*)
METHOD instantSort : CNM_CollectionInterfaces.CNM_ReturnTypes.SingleExecutionResult
VAR_INPUT
	(*The size of the list to be sorted*)
	size	: UDINT;
	(*Optional: the comparator that should be used for the sort. Must not be changed while sort is in process*)
	comparator	: CNM_CollectionInterfaces.CNM_AbstractObject.IComparator := 0;
END_VAR
VAR_IN_OUT
	(*The first element in the list, must be set on every call to current head of list.*)
	head	: CNM_CollectionInterfaces.IDoublyLinkedElement;
	(*The last element of the list after sorting, may be useful for doublelinked structures*)
	last	: CNM_CollectionInterfaces.IDoublyLinkedElement;
	(*the current version of the list, must change when the data in the list changes *)
	currentListVersion	: __XWORD;
END_VAR
VAR
	mergesThisRun 		:__XWORD;
	mergeSize			:__XWORD;
	mergeSizeLeft		:__XWORD;
	mergeSizeRight		:__XWORD;
	index				:__XWORD;
	leftElementToMerge	:CNM_CollectionInterfaces.IDoublyLinkedElement;
	rightElementToMerge	:CNM_CollectionInterfaces.IDoublyLinkedElement;
	sortComplete :BOOL := FALSE;
	comparesThisCycle	:__XWORD := 0;
END_VAR
VAR CONSTANT
	OBJECT_NOT_REFERENCED 	:__XWORD := 0;
END_VAR
THIS^.sorterHead := head;
THIS^.sorterLast := OBJECT_NOT_REFERENCED;
THIS^.setComparator(comparator);
mergeSize := 1;
WHILE NOT sortComplete DO
	IF THIS^.isObjectNull(leftElementToMerge) THEN 
		mergesThisRun := 0;	
		leftElementToMerge := THIS^.sorterHead;	
		THIS^.sorterHead := OBJECT_NOT_REFERENCED;
		THIS^.sorterLast := OBJECT_NOT_REFERENCED;		
	END_IF;
		
	//one run trought the list from left to right
	WHILE THIS^.isObjectValid(leftElementToMerge) DO
		mergesThisRun := mergesThisRun + 1;
		rightElementToMerge := leftElementToMerge;
		//place rightElement mergeSize steps right of leftElement
		mergeSizeLeft := 0;	
		FOR index := 0 TO mergeSize-1 DO
			mergeSizeLeft := mergeSizeLeft + 1;
			rightElementToMerge := rightElementToMerge.next;
			IF THIS^.isObjectNull(rightElementToMerge) THEN
				EXIT;
			END_IF
		END_FOR
		mergeSizeRight := mergeSize;
		
		THIS^.merge(	
			leftElement := leftElementToMerge,
			rightElement := rightElementToMerge,
			mergeSizeLeft := mergeSizeLeft,
			mergeSizeRight := mergeSizeRight,
			mergeHead := THIS^.sorterHead,
			mergeLast := THIS^.sorterLast,
			comparesThisCycle := comparesThisCycle
		);
		
		//set leftElementToMerge to first unmerged Element, as rightElementToMerge points to the Element behind the right Mergesection
		leftElementToMerge := rightElementToMerge;
	END_WHILE
	
	IF (mergesThisRun <= 1) AND THIS^.isObjectNull(leftElementToMerge) THEN
		sortComplete := TRUE;
	ELSIF THIS^.isObjectNull(leftElementToMerge) THEN
		mergeSize := mergeSize * 2;
	END_IF;
	
	head := THIS^.sorterHead;
	last := THIS^.sorterLast;

END_WHILE

currentListVersion := currentListVersion + 1;
instantSort := CNM_ReturnTypes.SingleExecutionResult.SUCCESS;
END_METHOD

(*

## Short summary

Does an inplace ordered Merge of two list sections, that are defined by their first object and the length of the section.
Merge is achived by updating the links of the elements.

.. <legal notes>

legal notes
=================
| SPDX-FileCopyrightText: © 2024 ekvip automation GmbH <info@ekvip.de>
| SPDX-License-Identifier: Apache-2.0
| For details check: Apache-2.0_

.. _Apache-2.0: https://www.apache.org/licenses/LICENSE-2.0

.. </legal notes>


**Return:** CNM_ReturnTypes.ExecutionState: the state of the merge, 
	SUCCESS if list is merged from left to right bound, 
	BUSY if list not completly merged, needs to be called again.

*)

METHOD PROTECTED merge
VAR_INPUT
	//how many elements are in the left section
	mergeSizeLeft 	:__XWORD;
	//how many elements are in the right section
	mergeSizeRight	:__XWORD;
END_VAR
VAR_IN_OUT
	//The updated head of the list that is beeing merged
	mergeHead			:CNM_CollectionInterfaces.IDoublyLinkedElement;
	//The updated last of the list that is beeing merged
	mergeLast			:CNM_CollectionInterfaces.IDoublyLinkedElement;
	//the first element of the left section
	leftElement			:CNM_CollectionInterfaces.IDoublyLinkedElement;
	// the first element of the right section
	rightElement		:CNM_CollectionInterfaces.IDoublyLinkedElement;
	//The amount of already performed compares this cycle
	comparesThisCycle :__XWORD;
END_VAR
VAR
	remainElementsLeft	:__XWORD := mergeSizeLeft;
	remainElementsRight	:__XWORD := mergeSizeRight;
	elementToMerge		:CNM_CollectionInterfaces.IDoublyLinkedElement;
	lastLeftElement	:CNM_CollectionInterfaces.IDoublyLinkedElement;
END_VAR
VAR CONSTANT
	OBJECT_NOT_REFERENCED :__XWORD := 0;
END_VAR
IF THIS^.isObjectValid(rightElement) THEN
	lastLeftElement := rightElement.previous;	
END_IF

//when remainElementsRight is greater 0, also check if currentRightElement is valid, may not be valid for the merge at end of the list
WHILE(remainElementsLeft > 0 AND_THEN remainElementsRight > 0 AND_THEN THIS^.isObjectValid(rightElement) ) DO
	//by comparing that way, when elements are equal, they are taken from left, making the sort Stable 
	IF THIS^.compareElements(rightElement.object,leftElement.object) = CNM_ReturnTypes.ComparationResult.SMALLER THEN
		elementToMerge := rightElement;
		rightElement := rightElement.next;
		remainElementsRight := remainElementsRight - 1;
	ELSE
		elementToMerge := leftElement;
		leftElement := leftElement.next;
		remainElementsLeft := remainElementsLeft - 1;
	END_IF;
	
	IF THIS^.isObjectNull(mergeHead) THEN
		mergeHead := elementToMerge;
	ELSE
		mergeLast.next := elementToMerge;
	END_IF;
	
	elementToMerge.previous := mergeLast;	
	mergeLast := elementToMerge;
	comparesThisCycle := comparesThisCycle+1;
END_WHILE

elementToMerge := SEL(
	remainElementsLeft > 0,
	rightElement,
	leftElement
);
moveRemainingElements(
	remainingElements := SEL(
		remainElementsLeft > 0,
		remainElementsRight,
		remainElementsLeft
	),
	elementToMerge := elementToMerge,
	mergeHead := mergeHead,
	mergeLast := mergeLast,
	lastRemainder := SEL(remainElementsLeft>0,OBJECT_NOT_REFERENCED,lastLeftElement),
	operationsCount := comparesThisCycle
);	

IF remainElementsRight > 0 AND_THEN THIS^.isObjectValid(rightElement) THEN
	rightElement := mergeLast.next;
ELSE
	mergeLast.next := rightElement;
END_IF

IF THIS^.isObjectValid(rightElement) THEN
	rightElement.previous := mergeLast;	
END_IF
END_METHOD

METHOD moveRemainingElements : BOOL
VAR_INPUT
	remainingElements :__XWORD;
	lastRemainder	:CNM_CollectionInterfaces.IDoublyLinkedElement;
END_VAR
VAR_IN_OUT
	elementToMerge	:CNM_CollectionInterfaces.IDoublyLinkedElement;
	mergeHead		:CNM_CollectionInterfaces.IDoublyLinkedElement;
	mergeLast		:CNM_CollectionInterfaces.IDoublyLinkedElement;
	
	operationsCount	:__XWORD;
END_VAR
//one side is empty, other needs to be "copied"
IF THIS^.isObjectNull(mergeHead) THEN
	mergeHead := elementToMerge;
ELSE
	mergeLast.next := elementToMerge;
END_IF;

elementToMerge.previous := mergeLast;	

IF THIS^.isObjectValid(lastRemainder) THEN
	// first and last of the remaining elements are know, so just move the whole section
	mergeLast := lastRemainder;
	operationsCount := operationsCount + 1;
ELSE
	//step over the leftover elements to figure out the last element of that section
	WHILE remainingElements > 0 AND_THEN THIS^.isObjectValid(elementToMerge) DO
		mergeLast := elementToMerge;	
		elementToMerge := elementToMerge.next;
		remainingElements := remainingElements - 1;
		operationsCount := operationsCount +1;
	END_WHILE
END_IF
END_METHOD

(*

## Short summary

This method sorts the data structure. 
It uses the passed Comperator to sort the structure.
This can take many cycles and should be called until the CNM_ReturnTypes.ExecutionState is no longer ``BUSY``.

.. <legal notes>

legal notes
=================
| SPDX-FileCopyrightText: © 2025 ekvip automation GmbH <info@ekvip.de>
| SPDX-License-Identifier: Apache-2.0
| For details check: Apache-2.0_

.. _Apache-2.0: https://www.apache.org/licenses/LICENSE-2.0

.. </legal notes>


**Return:** ``ABORTED``: While sort was pending,execute had a falling edge,
	``BUSY``: Sort is in progress
	``ERROR``: Sort was not able to finish (p.e. List changed) call sort(false) to reset
	``IDLE``: Currently no sort in progress
	``SUCCESS``: Sorting was finished 

*)
METHOD sort : CNM_ReturnTypes.SingleExecutionState
VAR_INPUT
	(*control bit to start or abort the sorting, needs to be active until the ExecutionState is SUCCESS*)
	execute	: BOOL;
	(*The size of the list to be sorted*)
	size :UDINT;
	(*the comparator that should be used for the sort. Must not be changed while sort is in process*)
	comparator	: CNM_AbstractObject.IComparator	:= 0;
END_VAR
VAR_IN_OUT
	(*The first element in the list, must be set on every call to current head of list.*)
	head :CNM_CollectionInterfaces.IDoublyLinkedElement;
	(*The last element of the list after sorting, may be useful for doublelinked structures*)
	last :CNM_CollectionInterfaces.IDoublyLinkedElement;
	(*the current version of the list, must change when the data in the list changes *)
	currentListVersion :__XWORD;
END_VAR
VAR_INST
	cycleManager 		:CNM_CycleManager.SimpleCycleManager;
	leftElementToMerge	:CNM_CollectionInterfaces.IDoublyLinkedElement;
	rightElementToMerge	:CNM_CollectionInterfaces.IDoublyLinkedElement;
	(*How many merges were made during traversing list from left to right*)
	mergesThisRun 		:__XWORD;
	mergeSize			:__XWORD;
	mergeSizeLeft		:__XWORD;
	mergeSizeRight		:__XWORD;
	index				:__XWORD;
	(* list version index, used to detect list changes during sorting *)
	lastListChangeIndex :__XWORD;
END_VAR
VAR
	comparesThisCycle	:__XWORD	:= 0;
END_VAR
VAR CONSTANT
	INIT	:DINT := CNM_ReturnTypes.DefaultSteps.STEP.INIT; 
	SUCCESS :DINT := CNM_ReturnTypes.DefaultSteps.STEP.SUCCESS;
	ERROR   :DINT := CNM_ReturnTypes.DefaultSteps.STEP.ERROR;
	RUN_SORT :DINT := INIT + 1;
	OBJECT_NOT_REFERENCED 	:__XWORD := 0;
END_VAR
cycleManager(execute := execute);
IF cycleManager.step.current > INIT THEN
	cycleManager.assert.bitNumber.x.valueIsEqualTo(
		currentValue := currentListVersion,
		expectedValue := lastListChangeIndex,
		message := 'List has changed during sort!'
	);
END_IF

CASE cycleManager.step.current OF
INIT:
	cycleManager.configuration.sequence.requireSuccessStep := FALSE;
	lastListChangeIndex := currentListVersion;
	THIS^.sorterHead := head;
	THIS^.sorterLast := OBJECT_NOT_REFERENCED;
	THIS^.setComparator(comparator);
	mergeSize := 1;
	cycleManager.proceedWith(
		step := SEL( (size > 1), SUCCESS, RUN_SORT)
	);
RUN_SORT:
	IF (currentListVersion <> lastListChangeIndex) THEN
		cycleManager.proceedWith(ERROR);
		sort := CNM_ReturnTypes.SingleExecutionState.ERROR;
		RETURN;
	ELSE
		IF THIS^.isObjectNull(leftElementToMerge) THEN 
			mergesThisRun := 0;	
			leftElementToMerge := THIS^.sorterHead;	
			THIS^.sorterHead := OBJECT_NOT_REFERENCED;
			THIS^.sorterLast := OBJECT_NOT_REFERENCED;		
		END_IF;
		
		//one run trought the list from left to right
		WHILE THIS^.isObjectValid(leftElementToMerge) DO
			//only do merge if it won't exceed comparelimit, but allow at least one merge per Cycle
			IF (comparesThisCycle > 0) AND_THEN (comparesThisCycle + mergeSizeLeft + mergeSizeRight > THIS^.upperCompareBound) THEN
				EXIT;
			END_IF
			mergesThisRun := mergesThisRun + 1;
			rightElementToMerge := leftElementToMerge;
			//place rightElement mergeSize steps right of leftElement
			mergeSizeLeft := 0;	
			FOR index := 0 TO mergeSize-1 DO
				mergeSizeLeft := mergeSizeLeft + 1;
				rightElementToMerge := rightElementToMerge.next;
				IF THIS^.isObjectNull(rightElementToMerge) THEN
					EXIT;
				END_IF
			END_FOR
			mergeSizeRight := mergeSize;
			
			THIS^.merge(	
				leftElement := leftElementToMerge,
				rightElement := rightElementToMerge,
				mergeSizeLeft := mergeSizeLeft,
				mergeSizeRight := mergeSizeRight,
				mergeHead := THIS^.sorterHead,
				mergeLast := THIS^.sorterLast,
				comparesThisCycle := comparesThisCycle
			);
			
			//set leftElementToMerge to first unmerged Element, as rightElementToMerge points to the Element behind the right Mergesection
			leftElementToMerge := rightElementToMerge;
		END_WHILE
	
		IF (mergesThisRun <= 1) AND THIS^.isObjectNull(leftElementToMerge) THEN
			cycleManager.proceedWith(SUCCESS);
		ELSIF THIS^.isObjectNull(leftElementToMerge) THEN
			mergeSize := mergeSize * 2;
		END_IF;
	
		head := THIS^.sorterHead;
		last := THIS^.sorterLast;
		
		lastListChangeIndex := currentListVersion := currentListVersion + 1;
	END_IF
END_CASE

sort := cycleManager.state;
END_METHOD

END_FUNCTION_BLOCK

// ---- Lists/Sorter/classes/AbstractLinkedListSorter.TcPOU
(*

## Short summary

Abstract base class for LinkedListSorters.
Handles the head and last properties as well as the clone.
.. <legal notes>

legal notes
=================
| SPDX-FileCopyrightText: © 2025 ekvip automation GmbH <info@ekvip.de>
| SPDX-License-Identifier: Apache-2.0
| For details check: Apache-2.0_

.. _Apache-2.0: https://www.apache.org/licenses/LICENSE-2.0

.. </legal notes>



*)

FUNCTION_BLOCK INTERNAL ABSTRACT AbstractLinkedListSorter EXTENDS AbstractListSorter IMPLEMENTS CNM_CollectionInterfaces.ILinkedListSorter
VAR
	sorterHead :CNM_CollectionInterfaces.IDoublyLinkedElement;
	sorterLast :CNM_CollectionInterfaces.IDoublyLinkedElement;
END_VAR

(*

## Short summary

This method sorts the data structure instantly in descending order within one call. 
Uses the passed Comparator or the compareTo of the contained Objects if no comparator is passed.

.. <legal notes>

legal notes
=================
| SPDX-FileCopyrightText: © 2022 ekvip automation GmbH <info@ekvip.de>
| SPDX-License-Identifier: Apache-2.0
| For details check: Apache-2.0_

.. _Apache-2.0: https://www.apache.org/licenses/LICENSE-2.0

.. </legal notes>


**Return:**``ERROR``: Sort was not able to finish 
	``SUCCESS``: Sorting was finished succesfully

*)
METHOD instantInverseSort : CNM_CollectionInterfaces.CNM_ReturnTypes.SingleExecutionResult
VAR_INPUT
	(*The size of the list to be sorted*)
	size	: UDINT;
	(*Optional: the comparator that should be used for the sort. Must not be changed while sort is in process*)
	comparator	: CNM_CollectionInterfaces.CNM_AbstractObject.IComparator := 0;
END_VAR
VAR_IN_OUT
	(*The first element in the list, must be set on every call to current head of list.*)
	head	: CNM_CollectionInterfaces.IDoublyLinkedElement;
	(*The last element of the list after sorting, may be useful for doublelinked structures*)
	last	: CNM_CollectionInterfaces.IDoublyLinkedElement;
	(*the current version of the list, must change when the data in the list changes *)
	currentListVersion	: __XWORD;
END_VAR
THIS^.reverseComparator.attachComparator(comparator);
THIS^.instantSort(
	size := size,
	comparator := THIS^.reverseComparator,
	head := head,
	last := last,
	currentListVersion := currentListVersion
);
END_METHOD

(*

## Short summary

This method sorts the data structure instantly within one call. 
Uses the passed Comparator or the compareTo of the contained Objects if no comparator is passed.

.. <legal notes>

legal notes
=================
| SPDX-FileCopyrightText: © 2022 ekvip automation GmbH <info@ekvip.de>
| SPDX-License-Identifier: Apache-2.0
| For details check: Apache-2.0_

.. _Apache-2.0: https://www.apache.org/licenses/LICENSE-2.0

.. </legal notes>


**Return:**``ERROR``: Sort was not able to finish 
	``SUCCESS``: Sorting was finished succesfully

*)
METHOD ABSTRACT instantSort : CNM_CollectionInterfaces.CNM_ReturnTypes.SingleExecutionResult
VAR_INPUT
	(*The size of the list to be sorted*)
	size	: UDINT;
	(*Optional: the comparator that should be used for the sort. Must not be changed while sort is in process*)
	comparator	: CNM_CollectionInterfaces.CNM_AbstractObject.IComparator := 0;
END_VAR
VAR_IN_OUT
	(*The first element in the list, must be set on every call to current head of list.*)
	head	: CNM_CollectionInterfaces.IDoublyLinkedElement;
	(*The last element of the list after sorting, may be useful for doublelinked structures*)
	last	: CNM_CollectionInterfaces.IDoublyLinkedElement;
	(*the current version of the list, must change when the data in the list changes *)
	currentListVersion	: __XWORD;
END_VAR
END_METHOD

(*

## Short summary

This method sorts the Sortable in the inverted order, so from great to low
.. <legal notes>

legal notes
=================
| SPDX-FileCopyrightText: © 2025 ekvip automation GmbH <info@ekvip.de>
| SPDX-License-Identifier: Apache-2.0
| For details check: Apache-2.0_

.. _Apache-2.0: https://www.apache.org/licenses/LICENSE-2.0

.. </legal notes>


**Return:** ``ABORTED``: While inverse was pending,execute had a falling edge,
	``BUSY``: Inverse is in progress
	``ERROR``: Inverse was not able to finish (p.e. List changed) call inverse(false) to reset
	``IDLE``: Currently invert is not in progress
	``SUCCESS``: Inversing was finished 
*)

METHOD inverseSort :CNM_ReturnTypes.SingleExecutionState;
VAR_INPUT
	(*control bit to start or abort the inverting, needs to be active until the ExecutionState is noz longer busy*)
	execute	:BOOL;
	(*The size of the list to be sorted*)
	size :UDINT;
END_VAR
VAR_INPUT
	(*the comparator that should be used for the sort. Must not be changed while sort is in process*)
	comparator :CNM_AbstractObject.IComparator := 0;
END_VAR
VAR_IN_OUT
	(*The first element in the list, must be set on every call to current head of list.*)
	head :CNM_CollectionInterfaces.IDoublyLinkedElement;
	(*The last element of the list after sorting, may be useful for doublelinked structures*)
	last :CNM_CollectionInterfaces.IDoublyLinkedElement;
	(*the current version of the list, must change when the data in the list changes *)
	currentListVersion :__XWORD;
END_VAR
THIS^.reverseComparator.attachComparator(comparator);
THIS^.sort(
	execute := execute,
	size := size,
	comparator := THIS^.reverseComparator,
	head := head,
	last := last,
	currentListVersion := currentListVersion
);
END_METHOD

(*

## Short summary

This method sorts the data structure. 
This can take many cycles and should be called until the CNM_ReturnTypes.ExecutionState is no longer ``BUSY``.
Call with execute := FALSE to initialize before sort.
.. <legal notes>

legal notes
=================
| SPDX-FileCopyrightText: © 2022 ekvip automation GmbH <info@ekvip.de>
| SPDX-License-Identifier: Apache-2.0
| For details check: Apache-2.0_

.. _Apache-2.0: https://www.apache.org/licenses/LICENSE-2.0

.. </legal notes>


**Return:** ``ABORTED``: While sort was pending,execute had a falling edge,
	``BUSY``: Sort is in progress
	``ERROR``: Sort was not able to finish (p.e. List changed) call sort(false) to reset
	``IDLE``: Currently no sort in progress
	``SUCCESS``: Sorting was finished 

*)

METHOD ABSTRACT sort :CNM_ReturnTypes.SingleExecutionState
VAR_INPUT
	(*control bit to start or abort the sorting, needs to be active until the ExecutionState is SUCCESS*)
	execute	:BOOL;
	(*The size of the list to be sorted*)
	size :UDINT;
	(*Optional: the comparator that should be used for the sort. Must not be changed while sort is in process*)
	comparator :CNM_AbstractObject.IComparator := 0;
END_VAR
VAR_IN_OUT
	(*The first element in the list, must be set on every call to current head of list.*)
	head :CNM_CollectionInterfaces.IDoublyLinkedElement;
	(*The last element of the list after sorting, may be useful for doublelinked structures*)
	last :CNM_CollectionInterfaces.IDoublyLinkedElement;
	(*the current version of the list, must change when the data in the list changes *)
	currentListVersion :__XWORD;
END_VAR
END_METHOD

END_FUNCTION_BLOCK

// ---- Utils/log2.TcPOU
(*

## Short summary

This function calculates the logarithmus dualis (ld or log_2). 
It uses [black magic](https://en.wikipedia.org/wiki/De_Bruijn_sequence). Actually it calculates the log2 and truncates it. 

.. <legal notes>

legal notes
=================
| SPDX-FileCopyrightText: © 2025 ekvip automation GmbH <info@ekvip.de>
| SPDX-License-Identifier: Apache-2.0
| For details check: Apache-2.0_

.. _Apache-2.0: https://www.apache.org/licenses/LICENSE-2.0

.. </legal notes>

*)

FUNCTION log2 : USINT
VAR_INPUT
	value :__UXINT(1..MAX_UXINT);
END_VAR
VAR
	architectureIndex :__XWORD;
	registerSize :USINT;
END_VAR
VAR CONSTANT
	MAX_UXINT :__UXINT := TO___UXINT(-1);
	DE_BRUIJN_SEQUENCE	:ARRAY[0..2] OF LWORD := [16#09AF ,16#077CB531, 16#022FDD63CC95386D];
	REGISTER_SIZE_IN_BYTES	:USINT := SIZEOF(__XWORD);
	DE_BRUIJN_LOOKUP :ARRAY[0..2] OF ARRAY[0..63] OF USINT := [
		[
			0, 1, 10, 2, 11, 14, 7, 3, 
        	12, 15, 8, 6, 13, 9, 5, 4
		],
		[
	    	0,  1, 28,  2, 29, 14, 24,  3, 
	    	30, 22, 20, 15, 25, 17,  4,  8, 
	    	31, 27, 13, 23, 21, 19, 16,  7, 
		    26, 12, 18,  6, 11,  5, 10,  9	
		],
		[
			0,  1,  2, 53,  3,  7, 54, 27,
			4, 38, 41,  8, 34, 55, 48, 28,
			62,  5, 39, 46, 44, 42, 22,  9,
			24, 35, 59, 56, 49, 18, 29, 11,
			63, 52,  6, 26, 37, 40, 33, 47,
			61, 45, 43, 21, 23, 58, 17, 10,
			51, 25, 36, 32, 60, 20, 57, 16,
			50, 31, 19, 15, 30, 14, 13, 12		
		]
	];
END_VAR

log2 := TO_USINT(-1);
RETURN(value <= 0);
architectureIndex := SHR(REGISTER_SIZE_IN_BYTES,2);
registerSize := SHL(REGISTER_SIZE_IN_BYTES,3);
value := value OR SHR(value, 1);
value := value OR SHR(value, 2);
value := value OR SHR(value, 4);
value := value OR SHR(value, 8);
value := SEL((REGISTER_SIZE_IN_BYTES > 2), value, (value OR SHR(value, 16)));
value := SEL((REGISTER_SIZE_IN_BYTES > 4), value, (value OR SHR(value, 32)));
IF (value = MAX_UXINT) THEN
	log2 := registerSize - 1;
ELSE
	log2 := DE_BRUIJN_LOOKUP[architectureIndex][
		SHR((value + 1) * DE_BRUIJN_SEQUENCE[architectureIndex],registerSize - (4 + architectureIndex))
	] - 1;
END_IF

END_FUNCTION

// ---- BinaryTree/Set/SetStrategyExecutor.TcPOU
FUNCTION_BLOCK INTERNAL SetStrategyExecutor EXTENDS CNM_AbstractObject.Object IMPLEMENTS CNM_CollectionInterfaces.ISetStrategy
VAR
	set :ISetHelper;
	instantExecutor :InstantSetStrategyExecutor;
END_VAR

(*

## Short summary

This abstract property returns the class name of the concrete object, 
which is useful for logging/debugging purpose.

.. <legal notes>

legal notes
=================
| SPDX-FileCopyrightText: © 2022 ekvip automation GmbH <info@ekvip.de>
| SPDX-License-Identifier: Apache-2.0
| For details check: Apache-2.0_

.. _Apache-2.0: https://www.apache.org/licenses/LICENSE-2.0

.. </legal notes>

*)
PROPERTY className : CNM_AbstractObject.ClassName
GET
className := 'CNM_Collections.SetStrategyExecutor';
END_GET
END_PROPERTY

(*

## Short summary

The constructor ``FB_init`` is needed to create an unique hash code.
The hash code is a pseudo random number create with a [xorshift](https://en.wikipedia.org/wiki/Xorshift) algorithm.
It can be overwritten on derivations, because it will be called implicit, ``SUPER^.FB_init()`` is not required.
For more information check: [Behavoir with derived function blocks](https://infosys.beckhoff.com/content/1033/tc3_plc_intro/5482088715.html?id=6983869892358031022).

.. <legal notes>

legal notes
=================
| SPDX-FileCopyrightText: © 2022 ekvip automation GmbH <info@ekvip.de>
| SPDX-License-Identifier: Apache-2.0
| For details check: Apache-2.0_

.. _Apache-2.0: https://www.apache.org/licenses/LICENSE-2.0

.. </legal notes>



*)
METHOD FB_init : BOOL
VAR_INPUT
	(* if TRUE, the retain variables are initialized (warm start / cold start)*)
	bInitRetains	: BOOL;
	(* if TRUE, the instance afterwards gets moved into the copy code (online change) *)
	bInCopyCode	: BOOL;
	(* the set which this executor will dispatch  *)
	set :ISetHelper;
END_VAR
THIS^.set := set;
THIS^.instantExecutor.assignSet(set);
END_METHOD

(*

## Short summary

Searches an object that is equal to the provided object in terms of the compareTo method (or a comparator provided by the parent).
 
.. <legal notes>

legal notes
=================
| SPDX-FileCopyrightText: © 2023 ekvip automation GmbH <info@ekvip.de>
| SPDX-License-Identifier: Apache-2.0
| For details check: Apache-2.0_

.. _Apache-2.0: https://www.apache.org/licenses/LICENSE-2.0

.. </legal notes>


**Return:** ``TRUE`` when an object that is equal is found, otherwise ``FALSE``

*)
METHOD getEqualObject : BOOL
VAR_INPUT
	(*The object to search for*)
	object	: CNM_CollectionInterfaces.CNM_AbstractObject.IObject;
END_VAR
VAR_OUTPUT
	(*The found object or null if not found*)
	foundObject	: CNM_CollectionInterfaces.CNM_AbstractObject.IObject;
END_VAR
getEqualObject := THIS^.set.getEqualObject(object := object, foundObject => foundObject);
END_METHOD

(*

## Short summary

This property returns a fluent interface for immediate (wihtin one call) operations of sets.

.. <legal notes>

legal notes
=================
| SPDX-FileCopyrightText: © 2025 ekvip automation GmbH <info@ekvip.de>
| SPDX-License-Identifier: Apache-2.0
| For details check: Apache-2.0_

.. _Apache-2.0: https://www.apache.org/licenses/LICENSE-2.0

.. </legal notes>

*)
PROPERTY instant : CNM_CollectionInterfaces.IInstantSetStrategy
GET
instant := THIS^.instantExecutor;
END_GET
END_PROPERTY

(*

## Short summary

overwrites the content of this set with the intersection of this set and the given set
Set intersection: Common elements between two sets.

**Example:**
Set A = {2, 3, 1, 4}
Set B = {3, 5, 6, 4}

Intersection of A and B: {3, 4}

.. <legal notes>

legal notes
=================
| SPDX-FileCopyrightText: © 2022 ekvip automation GmbH <info@ekvip.de>
| SPDX-License-Identifier: Apache-2.0
| For details check: Apache-2.0_

.. _Apache-2.0: https://www.apache.org/licenses/LICENSE-2.0

.. </legal notes>


**Return:** ``SUCCESS``: if intersect is complete
	``ABORTED``: execute has a falling edge during intersect,
	``BUSY``: Intersect is in Progress
	``ERROR``: the passed collection was not valid / contained invalid Elements

*)
METHOD intersect : CNM_CollectionInterfaces.CNM_ReturnTypes.SingleExecutionState
VAR_INPUT
	(*foreign set to intersect with*)
	set	: CNM_CollectionInterfaces.ISet;
	(*If intersect should be processed*)
	execute	: BOOL;
END_VAR
intersect := THIS^.set.intersect(set := set, execute := execute);
END_METHOD

(*

## Short summary

overwrites the content of this set with the union of this set and the given set
Set union: Combination of all elements from two sets.

**Example:**
Set A = {2, 3, 1, 4}
Set B = {3, 5, 6, 4}

Union of A and B: {1, 2, 3, 4, 5, 6}

.. <legal notes>

legal notes
=================
| SPDX-FileCopyrightText: © 2022 ekvip automation GmbH <info@ekvip.de>
| SPDX-License-Identifier: Apache-2.0
| For details check: Apache-2.0_

.. _Apache-2.0: https://www.apache.org/licenses/LICENSE-2.0

.. </legal notes>


**Return:** ``SUCCESS``: if merge completed, 
	``ABORTED``: execute has a falling edge during merge,
	``BUSY``: merge is in Progress
	``ERROR``: the passed collection where not valid / contained invalid Elements

*)
METHOD merge : CNM_CollectionInterfaces.CNM_ReturnTypes.SingleExecutionState
VAR_INPUT
	(*foreign set to merge with*)
	set	: CNM_CollectionInterfaces.ISet;
	(*If merge should be processed*)
	execute	: BOOL;
END_VAR
merge := THIS^.set.merge(set := set, execute := execute);
END_METHOD

(*

## Short summary

overwrites the content of this set with the set difference of this set and the given set
Set difference: Elements present in one set but not in the other.

**Example:**
Set A = {2, 3, 1, 4}
Set B = {3, 5, 6, 4}

Set difference (A - B): {1, 2}
Set difference (B - A): {5, 6}

.. <legal notes>

legal notes
=================
| SPDX-FileCopyrightText: © 2022 ekvip automation GmbH <info@ekvip.de>
| SPDX-License-Identifier: Apache-2.0
| For details check: Apache-2.0_

.. _Apache-2.0: https://www.apache.org/licenses/LICENSE-2.0

.. </legal notes>


**Return:** ``SUCCESS``: if insert could made, error if object was already in the tree,
	``ABORTED``: execute has a falling edge during insert,
	``BUSY``: Insert is in Progress
	``ERROR``: the passed collection where not valid / contained invalid Elements

*)
METHOD subtract : CNM_CollectionInterfaces.CNM_ReturnTypes.SingleExecutionState
VAR_INPUT
	(*foreign set to construct substraction*)
	set	: CNM_CollectionInterfaces.ISet;
	(*If substract should be processed*)
	execute	: BOOL;
END_VAR
subtract := THIS^.set.subtract(set := set, execute := execute);
END_METHOD

END_FUNCTION_BLOCK

// ---- BinaryTree/Set/InstantSetStrategyExecutor.TcPOU
FUNCTION_BLOCK INTERNAL InstantSetStrategyExecutor EXTENDS CNM_AbstractObject.Object IMPLEMENTS CNM_CollectionInterfaces.IInstantSetStrategy
VAR
	set :ISetHelper;
END_VAR

METHOD INTERNAL assignSet
VAR_INPUT
	set :ISetHelper;
END_VAR
THIS^.set := set;
END_METHOD

(*

## Short summary

This abstract property returns the class name of the concrete object, 
which is useful for logging/debugging purpose.

.. <legal notes>

legal notes
=================
| SPDX-FileCopyrightText: © 2022 ekvip automation GmbH <info@ekvip.de>
| SPDX-License-Identifier: Apache-2.0
| For details check: Apache-2.0_

.. _Apache-2.0: https://www.apache.org/licenses/LICENSE-2.0

.. </legal notes>

*)
PROPERTY className : CNM_AbstractObject.ClassName
GET
className := 'CNM_Collections.InstantSetExecutorStrategy';
END_GET
END_PROPERTY

(*

## Short summary

overwrites the content of this set with the intersection of this set and the given set
Set intersection: Common elements between two sets.

**Example:**
Set A = {2, 3, 1, 4}
Set B = {3, 5, 6, 4}

Intersection of A and B: {3, 4}

.. <legal notes>

legal notes
=================
| SPDX-FileCopyrightText: © 2022 ekvip automation GmbH <info@ekvip.de>
| SPDX-License-Identifier: Apache-2.0
| For details check: Apache-2.0_

.. _Apache-2.0: https://www.apache.org/licenses/LICENSE-2.0

.. </legal notes>


**Return:** ``SingleExecutionResult.SUCCESS``: if intersect is complete
	``SingleExecutionResult.ABORTED``: foreign set wasn't valid

*)
METHOD intersect : CNM_CollectionInterfaces.CNM_ReturnTypes.SingleExecutionResult
VAR_INPUT
	(*foreign set to intersect with*)
	set	: CNM_CollectionInterfaces.ISet;
END_VAR
intersect := THIS^.set.instantIntersect(set := set);
END_METHOD

(*

## Short summary

overwrites the content of this set with the union of this set and the given set
Set union: Combination of all elements from two sets.

**Example:**
Set A = {2, 3, 1, 4}
Set B = {3, 5, 6, 4}

Union of A and B: {1, 2, 3, 4, 5, 6}

.. <legal notes>

legal notes
=================
| SPDX-FileCopyrightText: © 2022 ekvip automation GmbH <info@ekvip.de>
| SPDX-License-Identifier: Apache-2.0
| For details check: Apache-2.0_

.. _Apache-2.0: https://www.apache.org/licenses/LICENSE-2.0

.. </legal notes>


**Return:** ``SUCCESS``: if merge completed
	```SingleExecutionResult.ABORTED``: foreign set wasn't valid

*)
METHOD merge : CNM_CollectionInterfaces.CNM_ReturnTypes.SingleExecutionResult
VAR_INPUT
	(*foreign set to merge with*)
	set	: CNM_CollectionInterfaces.ISet;
END_VAR
merge := THIS^.set.instantMerge(set := set);
END_METHOD

(*

## Short summary

overwrites the content of this set with the set difference of this set and the given set
Set difference: Elements present in one set but not in the other.

**Example:**
Set A = {2, 3, 1, 4}
Set B = {3, 5, 6, 4}

Set difference (A - B): {1, 2}
Set difference (B - A): {5, 6}

.. <legal notes>

legal notes
=================
| SPDX-FileCopyrightText: © 2022 ekvip automation GmbH <info@ekvip.de>
| SPDX-License-Identifier: Apache-2.0
| For details check: Apache-2.0_

.. _Apache-2.0: https://www.apache.org/licenses/LICENSE-2.0

.. </legal notes>


**Return:** ``SingleExecutionResult.SUCCESS``: if insert could made, error if object was already in the tree,
	```SingleExecutionResult.ABORTED``: foreign set wasn't valid

*)
METHOD subtract : CNM_CollectionInterfaces.CNM_ReturnTypes.SingleExecutionResult
VAR_INPUT
	(*foreign set to construct substraction*)
	set	: CNM_CollectionInterfaces.ISet;
END_VAR
subtract := THIS^.set.instantSubtract(set := set);
END_METHOD

END_FUNCTION_BLOCK

// ---- BinaryTree/Tree/TreeStrategyExecutor.TcPOU
FUNCTION_BLOCK TreeStrategyExecutor EXTENDS CNM_AbstractObject.Object IMPLEMENTS CNM_CollectionInterfaces.ITreeStrategy
VAR
	tree :ITreeHelper;
	instantExecutor :InstantTreeStrategyExecutor;
END_VAR

(*

## Short summary

This abstract property returns the class name of the concrete object, 
which is useful for logging/debugging purpose.

.. <legal notes>

legal notes
=================
| SPDX-FileCopyrightText: © 2022 ekvip automation GmbH <info@ekvip.de>
| SPDX-License-Identifier: Apache-2.0
| For details check: Apache-2.0_

.. _Apache-2.0: https://www.apache.org/licenses/LICENSE-2.0

.. </legal notes>

*)
PROPERTY className : CNM_AbstractObject.ClassName
GET
className := 'CNM_Collections.TreeStrategyExecutor';
END_GET
END_PROPERTY

(*

## Short summary

The constructor ``FB_init`` is needed to create an unique hash code.
The hash code is a pseudo random number create with a [xorshift](https://en.wikipedia.org/wiki/Xorshift) algorithm.
It can be overwritten on derivations, because it will be called implicit, ``SUPER^.FB_init()`` is not required.
For more information check: [Behavoir with derived function blocks](https://infosys.beckhoff.com/content/1033/tc3_plc_intro/5482088715.html?id=6983869892358031022).

.. <legal notes>

legal notes
=================
| SPDX-FileCopyrightText: © 2022 ekvip automation GmbH <info@ekvip.de>
| SPDX-License-Identifier: Apache-2.0
| For details check: Apache-2.0_

.. _Apache-2.0: https://www.apache.org/licenses/LICENSE-2.0

.. </legal notes>


*)
METHOD FB_init : BOOL
VAR_INPUT
	(* if TRUE, the retain variables are initialized (warm start / cold start)*)
	bInitRetains	: BOOL;
	(* if TRUE, the instance afterwards gets moved into the copy code (online change) *)
	bInCopyCode	: BOOL;
	(*the tree which this executor will dispatch to*)
	tree :ITreeHelper;
END_VAR
THIS^.tree := tree;
THIS^.instantExecutor.assignTree(tree);
END_METHOD

(*

## Short summary

A method to insert a single element into the tree.

.. <legal notes>

legal notes
=================
| SPDX-FileCopyrightText: © 2022 ekvip automation GmbH <info@ekvip.de>
| SPDX-License-Identifier: Apache-2.0
| For details check: Apache-2.0_

.. _Apache-2.0: https://www.apache.org/licenses/LICENSE-2.0

.. </legal notes>


**Return:** ``SUCCESS``: operation successful
	``ABORTED``: operation was aborted (implementation specific)
	``ERROR``: out of memory

*)
METHOD insert : CNM_CollectionInterfaces.CNM_ReturnTypes.SingleExecutionResult
VAR_INPUT
	(*the object that should be inserted*)
	object	: CNM_CollectionInterfaces.CNM_AbstractObject.IObject;
END_VAR
insert := THIS^.tree.insert(object := object);
END_METHOD

(*

## Short summary

This method inserts all elements of a collection into the tree.

If any value of the collection could not be inserted because of duplication, operation isn't aborted, 
insertion is tried for every element of the collection.

.. <legal notes>

legal notes
=================
| SPDX-FileCopyrightText: © 2025 ekvip automation GmbH <info@ekvip.de>
| SPDX-License-Identifier: Apache-2.0
| For details check: Apache-2.0_

.. _Apache-2.0: https://www.apache.org/licenses/LICENSE-2.0

.. </legal notes>


**Return:** ``SUCCESS``: if insert could be made
	``ABORTED``: execute has a falling edge during insert,
	``BUSY``: Insert is in Progress
	``ERROR``: the passed collection where not valid / contained invalid Elements
	``IDLE``: method was never started

*)
METHOD insertCollection : CNM_CollectionInterfaces.CNM_ReturnTypes.SingleExecutionState
VAR_INPUT
	(*The collection that should be inserted*)
	collection	: CNM_CollectionInterfaces.ICollection;
	(*If insert should be processed*)
	execute	: BOOL;
END_VAR
insertCollection := THIS^.tree.insertCollection(collection := collection, execute := execute);
END_METHOD

(*

## Short summary

This property returns a fluent interface for immediate (wihtin one call) operations of tree.

.. <legal notes>

legal notes
=================
| SPDX-FileCopyrightText: © 2025 ekvip automation GmbH <info@ekvip.de>
| SPDX-License-Identifier: Apache-2.0
| For details check: Apache-2.0_

.. _Apache-2.0: https://www.apache.org/licenses/LICENSE-2.0

.. </legal notes>

*)
PROPERTY instant : CNM_CollectionInterfaces.IInstantTreeStrategy
GET
instant := THIS^.instantExecutor;
END_GET
END_PROPERTY

(*

## Short summary

Function to remove an object from the tree

.. <legal notes>

legal notes
=================
| SPDX-FileCopyrightText: © 2022 ekvip automation GmbH <info@ekvip.de>
| SPDX-License-Identifier: Apache-2.0
| For details check: Apache-2.0_

.. _Apache-2.0: https://www.apache.org/licenses/LICENSE-2.0

.. </legal notes>


**Return:** ``SUCCESS``: if remove could be made
	``ABORTED``: if object wasn't in the tree
	``ERROR``: if object wasn't valid

*)
METHOD remove : CNM_CollectionInterfaces.CNM_ReturnTypes.SingleExecutionResult
VAR_INPUT
	(* The object that should be removed *)
	object	: CNM_CollectionInterfaces.CNM_AbstractObject.IObject;
END_VAR
remove := THIS^.tree.remove(object := object);
END_METHOD

END_FUNCTION_BLOCK

// ---- BinaryTree/Tree/InstantTreeStrategyExecutor.TcPOU
FUNCTION_BLOCK InstantTreeStrategyExecutor EXTENDS CNM_AbstractObject.Object IMPLEMENTS CNM_CollectionInterfaces.IInstantTreeStrategy
VAR
	tree :ITreeHelper;
END_VAR

METHOD INTERNAL assignTree
VAR_INPUT
	tree :ITreeHelper;
END_VAR
THIS^.tree := tree;
END_METHOD

(*

## Short summary

This abstract property returns the class name of the concrete object, 
which is useful for logging/debugging purpose.

.. <legal notes>

legal notes
=================
| SPDX-FileCopyrightText: © 2022 ekvip automation GmbH <info@ekvip.de>
| SPDX-License-Identifier: Apache-2.0
| For details check: Apache-2.0_

.. _Apache-2.0: https://www.apache.org/licenses/LICENSE-2.0

.. </legal notes>

*)
PROPERTY className : CNM_AbstractObject.ClassName
GET
className := 'CNM_Collections.InstantTreeStrategyExecutor';
END_GET
END_PROPERTY

(*

## Short summary

This method inserts all elements of a collection into the tree
This takes only one cycle 

.. <legal notes>

legal notes
=================
| SPDX-FileCopyrightText: © 2022 ekvip automation GmbH <info@ekvip.de>
| SPDX-License-Identifier: Apache-2.0
| For details check: Apache-2.0_

.. _Apache-2.0: https://www.apache.org/licenses/LICENSE-2.0

.. </legal notes>


**Return:** ``SingleExecutionResult.SUCCESS``: operation successful
	``SingleExecutionResult.ERROR``: out of memory
	``SingleExecutionResult.ABORTED``: collection to insert wasn't valid

*)
METHOD insertCollection : CNM_CollectionInterfaces.CNM_ReturnTypes.SingleExecutionResult
VAR_INPUT
	(*The collection that should be inserted*)
	collection	: CNM_CollectionInterfaces.ICollection;
END_VAR
insertCollection := THIS^.tree.instantInsertCollection(collection := collection);
END_METHOD

END_FUNCTION_BLOCK

// ---- BinaryTree/classes/BalancedBinarySearchTreeNode.TcPOU
(*

## Short summary

Class for a balanced, binary, search tree node

.. <legal notes>

legal notes
=================
| SPDX-FileCopyrightText: © 2022 ekvip automation GmbH <info@ekvip.de>
| SPDX-License-Identifier: Apache-2.0
| For details check: Apache-2.0_

.. _Apache-2.0: https://www.apache.org/licenses/LICENSE-2.0

.. </legal notes>



*)
{attribute 'enable_dynamic_creation'}
FUNCTION_BLOCK BalancedBinarySearchTreeNode EXTENDS AbstractDisposableContainer IMPLEMENTS CNM_CollectionInterfaces.IBalancedBinarySearchTreeNode
VAR
	nodevalue 			:CNM_AbstractObject.IObject;
	left 				:CNM_CollectionInterfaces.IBinaryTreeNode;
	right				:CNM_CollectionInterfaces.IBinaryTreeNode;
	nodebalance			:CNM_CollectionInterfaces.TreeBalance;
END_VAR

(*

## Short summary

This property represents the balance state for this node, for details see ``Tree_Balance`` from Interfacelib

.. <legal notes>

legal notes
=================
| SPDX-FileCopyrightText: © 2022 ekvip automation GmbH <info@ekvip.de>
| SPDX-License-Identifier: Apache-2.0
| For details check: Apache-2.0_

.. _Apache-2.0: https://www.apache.org/licenses/LICENSE-2.0

.. </legal notes>

*)

PROPERTY balance :CNM_CollectionInterfaces.TreeBalance
GET
balance := THIS^.nodebalance;
END_GET
SET
THIS^.nodebalance := balance;
END_SET
END_PROPERTY


(*

## Short summary

This abstract property returns the class name of the concrete object, 
which is useful to check the class name for ``__DELETE``.

.. <legal notes>

legal notes
=================
| SPDX-FileCopyrightText: © 2022 ekvip automation GmbH <info@ekvip.de>
| SPDX-License-Identifier: Apache-2.0
| For details check: Apache-2.0_

.. _Apache-2.0: https://www.apache.org/licenses/LICENSE-2.0

.. </legal notes>

*)
PROPERTY className :CNM_AbstractObject.ClassName
GET
className := 'CNM_Collections.BalancedBinarySearchTreeNode';
END_GET
END_PROPERTY

(*

## Short summary

This method is called in the destruct method and is intended to zero all references and interfaces that should not be destructed. 
To delete the collection with all its contents, use deepDestruct() instead of destruct().

.. <legal notes>

legal notes
=================
| SPDX-FileCopyrightText: © 2025 ekvip automation GmbH <info@ekvip.de>
| SPDX-License-Identifier: Apache-2.0
| For details check: Apache-2.0_

.. _Apache-2.0: https://www.apache.org/licenses/LICENSE-2.0

.. </legal notes>

*)
METHOD PROTECTED clearContents
VAR CONSTANT
	(* NULL is a constant which is always 0 *)
	NULL						:__XWORD	:= 0;
END_VAR
THIS^.left := NULL;
THIS^.right := NULL;
THIS^.nodevalue := NULL;
END_METHOD


(*

## Short summary

This method is used to create a new instance
of the object which has the same internal state as the object.
If the object is a container class, the content objects
are not cloned, for this there is the method ``ICloneable.deepClone``.

If an object does not support cloning the return value is
``CNM_ReturnTypes.CloneResult.CLONE_IS_NOT_SUPPORTED``.

If there is not enough memory or the cloning fails, because the
attribute enable dynamic creation was forgotten, the return value is 
``CNM_ReturnTypes.CloneResult.FAILED``.

Only if the return value is ``CNM_ReturnTypes.CloneResult.SUCCESS``
the output ``clonedObject`` points to the new object
otherwise ``clonedObject`` is NULL.  

.. <legal notes>

legal notes
=================
| SPDX-FileCopyrightText: © 2022 ekvip automation GmbH <info@ekvip.de>
| SPDX-License-Identifier: Apache-2.0
| For details check: Apache-2.0_

.. _Apache-2.0: https://www.apache.org/licenses/LICENSE-2.0

.. </legal notes>


**Return:** ``CNM_ReturnTypes.CloneResult.SUCCESS``: new object clone was created,
	``CNM_ReturnTypes.CloneResult.FAILED``: object clone failed
	``CNM_ReturnTypes.CloneResult.CLONE_IS_NOT_SUPPORTED``: object does not support cloning

*)
METHOD clone :CNM_AbstractObject.CNM_ReturnTypes.CloneResult
VAR_OUTPUT
	(* new object instance or NULL if somthing went wrong *)
	clonedObject			:CNM_AbstractObject.IObject;
END_VAR
VAR
	newTreeNode 			:POINTER TO BalancedBinarySearchTreeNode;
	newChildObject			:CNM_AbstractObject.IObject;
	newChildNode 			:CNM_CollectionInterfaces.IBinaryTreeNode;
END_VAR
VAR CONSTANT
	OBJECT_NOT_REFERENCED 	:__XWORD := 0;
END_VAR
newTreeNode := __NEW(
	BalancedBinarySearchTreeNode(
		value := THIS^.object,
		left := OBJECT_NOT_REFERENCED,
		right := OBJECT_NOT_REFERENCED
	)
);
IF (newTreeNode = 0) THEN
	clone := CNM_ReturnTypes.CloneResult.FAILED;
	RETURN;
ELSIF THIS^.isObjectValid(newTreeNode^) THEN
	clone := CNM_ReturnTypes.CloneResult.SUCCESS;
	IF THIS^.isObjectValid(THIS^.left) THEN
		clone := THIS^.left.clone(clonedObject => newChildObject);
		__QUERYINTERFACE(newCHildObject,newChildNode);
		newTreeNode^.leftChild := newChildNode;
	END_IF
	IF THIS^.isObjectValid(THIS^.right) AND clone = CNM_ReturnTypes.CloneResult.SUCCESS THEN
		clone := THIS^.right.clone(clonedObject => newChildObject);
		__QUERYINTERFACE(newCHildObject,newChildNode);
		newTreeNode^.rightChild := newChildNode;
	END_IF
	clonedObject := newTreeNode^;
	RETURN(clone = CNM_ReturnTypes.CloneResult.SUCCESS);		
ELSE
	clone := CNM_ReturnTypes.CloneResult.FAILED;
END_IF

//clone wasn't success, clean up
IF THIS^.isObjectValid(newTreeNode^) THEN
	THIS^.destructNodeAndAllChilds(newTreeNode^);
	clonedObject := OBJECT_NOT_REFERENCED;
END_IF
END_METHOD


(*

## Short summary

This method compares a foreign object with the own one, this is needed for sort orders.

.. <legal notes>

legal notes
=================
| SPDX-FileCopyrightText: © 2022 ekvip automation GmbH <info@ekvip.de>
| SPDX-License-Identifier: Apache-2.0
| For details check: Apache-2.0_

.. _Apache-2.0: https://www.apache.org/licenses/LICENSE-2.0

.. </legal notes>


**Return:** ``SMALLER``: ``THIS`` precedes in order,
	``EQUAL``: ``THIS`` and ``object`` at the same position in order,
	``GREATER``: ``THIS`` is after in order.
	Checkout the library CNM_ReturnTypes.

*)
METHOD compareTo :CNM_AbstractObject.CNM_ReturnTypes.ComparationResult
VAR_INPUT
	(* foreign object to compare*)
	object	:CNM_AbstractObject.IObject;
END_VAR
VAR 
	node 	:CNM_CollectionInterfaces.IBinaryTreeNode;
	compareObject	:CNM_AbstractObject.IObject;
END_VAR
compareTo := CNM_AbstractObject.CNM_ReturnTypes.ComparationResult.GREATER;
IF THIS^.isObjectValid(object) THEN 
	IF(__QUERYINTERFACE(object,node)) THEN
		compareObject := node.object;
	ELSE
		compareObject := object;
	END_IF
	
	IF(THIS^.isObjectValid(THIS^.object))THEN     
		compareTo := THIS^.object.compareTo(compareObject);
	END_IF
END_IF
END_METHOD


(*

## Short summary

This method is used to create a new instance
of the object which has the same internal state as the object.
If the object is a container class, the references to the content objects
are cloned too.

If an object does not support cloning the return value is
``CNM_ReturnTypes.CloneResult.CLONE_IS_NOT_SUPPORTED``.

If there is not enough memory or the cloning fails because the
attribute enable dynamic creation was forgotten the return value is 
``CNM_ReturnTypes.CloneResult.FAILED``.
If something goes wrong, then this method must clean up everything
that has been cloned and free the memory again.
**The deepClone either works completely, or not at all**

Only if the return value is ``CNM_ReturnTypes.CloneResult.SUCCESS``
the output ``clonedObject`` points to the new object
otherwise ``clonedObject`` is NULL.  

.. <legal notes>

legal notes
=================
| SPDX-FileCopyrightText: © 2022 ekvip automation GmbH <info@ekvip.de>
| SPDX-License-Identifier: Apache-2.0
| For details check: Apache-2.0_

.. _Apache-2.0: https://www.apache.org/licenses/LICENSE-2.0

.. </legal notes>


**Return:** ``CNM_ReturnTypes.CloneResult.SUCCESS``: new object clone was created,
	``CNM_ReturnTypes.CloneResult.FAILED``: object clone failed
	``CNM_ReturnTypes.CloneResult.CLONE_IS_NOT_SUPPORTED``: object does not support deep cloning

*)
METHOD deepClone :CNM_AbstractObject.CNM_ReturnTypes.CloneResult
VAR_OUTPUT
	(* new object instance or NULL if somthing went wrong *)
	clonedObject			:CNM_AbstractObject.IObject;
END_VAR
VAR
	newTreeNode 			:POINTER TO BalancedBinarySearchTreeNode;
	newChildObject			:CNM_AbstractObject.IObject;
	newChildNode 			:CNM_CollectionInterfaces.IBinaryTreeNode;
	newContent				:CNM_AbstractObject.IObject;
	cloneResult 			:CNM_ReturnTypes.CloneResult;
END_VAR
VAR CONSTANT
	OBJECT_NOT_REFERENCED 	:__XWORD := 0;
END_VAR
IF ( NOT THIS^.isObjectValid(THIS^.object)) THEN
	deepClone := CNM_ReturnTypes.CloneResult.FAILED;
	RETURN;
ELSIF ((cloneResult := THIS^.object.deepClone(clonedObject => newContent)) <> CNM_ReturnTypes.CloneResult.SUCCESS) THEN
	deepClone := cloneResult;
	RETURN;
END_IF

newTreeNode := __NEW(
	BalancedBinarySearchTreeNode(
		value := newContent,
		left := OBJECT_NOT_REFERENCED,
		right := OBJECT_NOT_REFERENCED
	)
);
IF (newTreeNode = 0) THEN
	newContent.deepDestruct();
	deepClone := CNM_ReturnTypes.CloneResult.FAILED;
	RETURN;
ELSIF THIS^.isObjectValid(newTreeNode^) THEN
	deepClone := CNM_ReturnTypes.CloneResult.SUCCESS;
	IF THIS^.isObjectValid(THIS^.left) THEN
		deepClone := THIS^.left.deepClone(clonedObject => newChildObject);
		__QUERYINTERFACE(newCHildObject,newChildNode);
		newTreeNode^.leftChild := newChildNode;
	END_IF
	IF THIS^.isObjectValid(THIS^.right) AND deepClone = CNM_ReturnTypes.CloneResult.SUCCESS THEN
		deepClone := THIS^.right.deepClone(clonedObject => newChildObject);
		__QUERYINTERFACE(newCHildObject,newChildNode);
		newTreeNode^.rightChild := newChildNode;
	END_IF
	clonedObject := newTreeNode^;
	RETURN(deepClone = CNM_ReturnTypes.CloneResult.SUCCESS);		
ELSE
	deepClone := CNM_ReturnTypes.CloneResult.FAILED;
END_IF

//deepclone wasn't success, clean up

IF THIS^.isObjectValid(newTreeNode^) THEN
	newTreeNode^.deepDestruct();
	clonedObject := OBJECT_NOT_REFERENCED;
ELSIF THIS^.isObjectValid(newContent) THEN
	newContent.deepDestruct();
END_IF
END_METHOD

(*

## Short summary

destructs / deepdestructs all nodes in the subtrees of a specified node and this node

.. <legal notes>

legal notes
=================
| SPDX-FileCopyrightText: © 2022 ekvip automation GmbH <info@ekvip.de>
| SPDX-License-Identifier: Apache-2.0
| For details check: Apache-2.0_

.. _Apache-2.0: https://www.apache.org/licenses/LICENSE-2.0

.. </legal notes>



*)

METHOD PROTECTED FINAL destructNodeAndAllChilds
VAR_INPUT
	(*the node that should be destructed with all it's childs*)
	node							:CNM_CollectionInterfaces.IBinaryTreeNode;
END_VAR
VAR CONSTANT
	OBJECT_NOT_REFERENCED			:__XWORD := 0;
END_VAR
RETURN(THIS^.isObjectNull(node));
IF THIS^.isObjectValid(node.leftChild) THEN
	THIS^.destructNodeAndAllChilds(node := node.leftChild);
	node.leftChild := OBJECT_NOT_REFERENCED;
END_IF
IF THIS^.isObjectValid(node.rightChild) THEN
	THIS^.destructNodeAndAllChilds(node := node.rightChild);
	node.rightChild := OBJECT_NOT_REFERENCED;
END_IF
node.destruct();
END_METHOD

(*

## Short summary

Mark the object as deleted, as it staiys in the memory.

.. <legal notes>

legal notes
=================
| SPDX-FileCopyrightText: © 2022 ekvip automation GmbH <info@ekvip.de>
| SPDX-License-Identifier: Apache-2.0
| For details check: Apache-2.0_

.. _Apache-2.0: https://www.apache.org/licenses/LICENSE-2.0

.. </legal notes>

*)
METHOD FB_Exit : BOOL
VAR_INPUT
	(* TRUE: the exit method is called in order to leave the instance which will be copied afterwards (online change).*)
	bInCopyCode	: BOOL;
END_VAR
IF THIS^.isObjectValid(THIS^.nodevalue) THEN
	THIS^.nodevalue.deepDestruct();
END_IF
IF THIS^.isObjectValid(THIS^.left) THEN
	THIS^.left.deepDestruct();
END_IF
IF THIS^.isObjectValid(THIS^.right) THEN
	THIS^.right.deepDestruct();
END_IF
END_METHOD

(*

## Short summary

The constructor ``FB_init`` is needed to create an unique hash code.
The hash code is a pseudo random number create with a [xorshift](https://en.wikipedia.org/wiki/Xorshift) algorithm.
It can be overwritten on derivations, because it will be called implicit, ``SUPER^.FB_init()`` is not required.
For more information check: [Behavoir with derived function blocks](https://infosys.beckhoff.com/content/1033/tc3_plc_intro/5482088715.html?id=6983869892358031022).

.. <legal notes>

legal notes
=================
| SPDX-FileCopyrightText: © 2022 ekvip automation GmbH <info@ekvip.de>
| SPDX-License-Identifier: Apache-2.0
| For details check: Apache-2.0_

.. _Apache-2.0: https://www.apache.org/licenses/LICENSE-2.0

.. </legal notes>



*)

METHOD FB_init : BOOL
VAR_INPUT
	(* if TRUE, the retain variables are initialized (warm start / cold start)*)
	bInitRetains	:BOOL;
	(* if TRUE, the instance afterwards gets moved into the copy code (online change) *)
	bInCopyCode		:BOOL;  
	value 						:CNM_AbstractObject.IObject;
	left 						:CNM_CollectionInterfaces.IBalancedBinarySearchTreeNode;
	right 						:CNM_CollectionInterfaces.IBalancedBinarySearchTreeNode;
END_VAR
VAR
	{attribute 'hide'}
	newHashstate3				:CNM_AbstractObject.Hashcode;
END_VAR
VAR CONSTANT
	{attribute 'hide'}
	NUMBER_OF_LEFT_SHIFTS		:UINT	:= 17;
	{attribute 'hide'}
	NUMBER_OF_LEFT_ROTATIONS	:UINT   := 45;
	OBJECT_NOT_REFERENCED 		:__XWORD := 0;
END_VAR
THIS^.object := value;
THIS^.right := right;
THIS^.left := left;
END_METHOD

(*

## Short summary

This property points to the left child of a binary tree node.
The injected node will be deleted within the deepdestruct context. 

.. <legal notes>

legal notes
=================
| SPDX-FileCopyrightText: © 2022 ekvip automation GmbH <info@ekvip.de>
| SPDX-License-Identifier: Apache-2.0
| For details check: Apache-2.0_

.. _Apache-2.0: https://www.apache.org/licenses/LICENSE-2.0

.. </legal notes>

*)

PROPERTY leftChild :CNM_CollectionInterfaces.IBinaryTreeNode
GET
leftChild := THIS^.left;
END_GET
SET
VAR CONSTANT
	OBJECT_NOT_REFERENCED :__XWORD := 0;
END_VAR
IF THIS^.isObjectValid(leftChild) THEN
	THIS^.left := leftChild;
ELSE
	THIS^.left := OBJECT_NOT_REFERENCED;
END_IF
END_SET
END_PROPERTY

(*

## Short summary

The property points to the content of the treenode. 
The object will be deleted within the deepdestruct context.

**Attention:** object is not allowed to be null since collections aren't allowed to contain null objects!

.. <legal notes>

legal notes
=================
| SPDX-FileCopyrightText: © 2022 ekvip automation GmbH <info@ekvip.de>
| SPDX-License-Identifier: Apache-2.0
| For details check: Apache-2.0_

.. _Apache-2.0: https://www.apache.org/licenses/LICENSE-2.0

.. </legal notes>

*)

PROPERTY object :CNM_AbstractObject.IObject
GET
object := THIS^.nodevalue;
END_GET
SET
THIS^.nodevalue := object;
END_SET
END_PROPERTY


(*

## Short summary

This property points to the right child of an binarytreeenode.
The injected node will be deleted within the deepdestruct context.

.. <legal notes>

legal notes
=================
| SPDX-FileCopyrightText: © 2022 ekvip automation GmbH <info@ekvip.de>
| SPDX-License-Identifier: Apache-2.0
| For details check: Apache-2.0_

.. _Apache-2.0: https://www.apache.org/licenses/LICENSE-2.0

.. </legal notes>

*)
PROPERTY rightChild :CNM_CollectionInterfaces.IBinaryTreeNode
GET
rightChild := THIS^.right;
END_GET
SET
VAR
END_VAR
VAR CONSTANT
	OBJECT_NOT_REFERENCED : __XWORD := 0;
END_VAR
IF THIS^.isObjectValid(rightChild) THEN
	  THIS^.right := rightChild;
ELSE
	  THIS^.right := OBJECT_NOT_REFERENCED;
END_IF
END_SET
END_PROPERTY

END_FUNCTION_BLOCK

// ---- Lists/LinkedList/classes/DoublyLinkedElement.TcPOU
(*

## Short summary

Implementation of IDoublyLinkElement.
Does not allow NULL as object.


.. <legal notes>

legal notes
=================
| SPDX-FileCopyrightText: © 2022 ekvip automation GmbH <info@ekvip.de>
| SPDX-License-Identifier: Apache-2.0
| For details check: Apache-2.0_

.. _Apache-2.0: https://www.apache.org/licenses/LICENSE-2.0

.. </legal notes>



*)
{attribute 'hide'}
{attribute 'enable_dynamic_creation'}
FUNCTION_BLOCK INTERNAL DoublyLinkedElement EXTENDS AbstractDisposableContainer IMPLEMENTS CNM_CollectionInterfaces.IDoublyLinkedElement
VAR
	nextElement 	:CNM_CollectionInterfaces.IDoublyLinkedElement;
	previousElement :CNM_CollectionInterfaces.IDoublyLinkedElement;
	dataObject 		:CNM_AbstractObject.IObject;
END_VAR

(*

## Short summary

This abstract property returns the class name of the concrete object, 
which is useful to check the class name for ``__DELETE``.

.. <legal notes>

legal notes
=================
| SPDX-FileCopyrightText: © 2022 ekvip automation GmbH <info@ekvip.de>
| SPDX-License-Identifier: Apache-2.0
| For details check: Apache-2.0_

.. _Apache-2.0: https://www.apache.org/licenses/LICENSE-2.0

.. </legal notes>

*)
PROPERTY className : CNM_AbstractObject.ClassName
GET
className := 'CNM_Collections.DoublyLinkedElement';
END_GET
END_PROPERTY

(*

## Short summary

This method is called in the destruct method and is intended to zero all references and interfaces that should not be destructed. 
To delete the collection with all its contents, use deepDestruct() instead of destruct().

.. <legal notes>

legal notes
=================
| SPDX-FileCopyrightText: © 2025 ekvip automation GmbH <info@ekvip.de>
| SPDX-License-Identifier: Apache-2.0
| For details check: Apache-2.0_

.. _Apache-2.0: https://www.apache.org/licenses/LICENSE-2.0

.. </legal notes>

*)
METHOD PROTECTED clearContents
VAR CONSTANT
	(* NULL is a constant which is always 0 *)
	NULL				:__XWORD := 0;
END_VAR
THIS^.dataObject := NULL;
END_METHOD

(*

## Short summary

This method is called in the deepDestruct method and is intended to destruct all contained Objects of the collection. 
To delete only the collection without deleting all its contents, use destruct() instead of deepDestruct().

.. <legal notes>

legal notes
=================
| SPDX-FileCopyrightText: © 2025 ekvip automation GmbH <info@ekvip.de>
| SPDX-License-Identifier: Apache-2.0
| For details check: Apache-2.0_

.. _Apache-2.0: https://www.apache.org/licenses/LICENSE-2.0

.. </legal notes>

*)

METHOD PROTECTED destructContents
IF (THIS^.isObjectValid(THIS^.dataObject)) THEN
	THIS^.dataObject.deepDestruct();
END_IF
END_METHOD

(*

## Short summary

Mark the object as deleted, as it staiys in the memory.

.. <legal notes>

legal notes
=================
| SPDX-FileCopyrightText: © 2022 ekvip automation GmbH <info@ekvip.de>
| SPDX-License-Identifier: Apache-2.0
| For details check: Apache-2.0_

.. _Apache-2.0: https://www.apache.org/licenses/LICENSE-2.0

.. </legal notes>

*)
METHOD FB_Exit : BOOL
VAR_INPUT
	(* TRUE: the exit method is called in order to leave the instance which will be copied afterwards (online change).*)
	bInCopyCode	: BOOL;
END_VAR
IF (THIS^.isObjectValid(THIS^.dataObject)) THEN
	THIS^.dataObject.deepDestruct();
END_IF
END_METHOD

(*

## Short summary

The constructor ``FB_init`` is needed to create an unique hash code.
The hash code is a pseudo random number create with a [xorshift](https://en.wikipedia.org/wiki/Xorshift) algorithm.
It can be overwritten on derivations, because it will be called implicit, ``SUPER^.FB_init()`` is not required.
For more information check: [Behavoir with derived function blocks](https://infosys.beckhoff.com/content/1033/tc3_plc_intro/5482088715.html?id=6983869892358031022).

.. <legal notes>

legal notes
=================
| SPDX-FileCopyrightText: © 2022 ekvip automation GmbH <info@ekvip.de>
| SPDX-License-Identifier: Apache-2.0
| For details check: Apache-2.0_

.. _Apache-2.0: https://www.apache.org/licenses/LICENSE-2.0

.. </legal notes>



*)

METHOD FB_init : BOOL
VAR_INPUT
	(* if TRUE, the retain variables are initialized (warm start / cold start)*)
	bInitRetains	:BOOL;
	(* if TRUE, the instance afterwards gets moved into the copy code (online change) *)
	bInCopyCode		:BOOL;  
	content 			:CNM_AbstractObject.IObject;
	next 	:CNM_CollectionInterfaces.IDoublyLinkedElement;
	previous :CNM_CollectionInterfaces.IDoublyLinkedElement;
END_VAR
VAR
	{attribute 'hide'}
	newHashstate3		:CNM_AbstractObject.Hashcode;
END_VAR
VAR CONSTANT
	{attribute 'hide'}
	NUMBER_OF_LEFT_SHIFTS		:UINT	:= 17;
	{attribute 'hide'}
	NUMBER_OF_LEFT_ROTATIONS	:UINT   := 45;
END_VAR
THIS^.object := content;
THIS^.next := next;
THIS^.previous := previous;
END_METHOD


(*

## Short summary

This property returns the next element that is linked to this element. Next element previous should be this object.
Next is not effected by deepdestruct.

.. <legal notes>

legal notes
=================
| SPDX-FileCopyrightText: © 2022 ekvip automation GmbH <info@ekvip.de>
| SPDX-License-Identifier: Apache-2.0
| For details check: Apache-2.0_

.. _Apache-2.0: https://www.apache.org/licenses/LICENSE-2.0

.. </legal notes>

*)
PROPERTY next : CNM_CollectionInterfaces.IDoublyLinkedElement
GET
next := THIS^.nextElement;
END_GET
SET
THIS^.nextElement := next;
END_SET
END_PROPERTY


(*

## Short summary

This property returns `CNM_AbstractObject.IObject` that represents the data of this element.
The passed object will be destroyed in deepDestruct.

.. <legal notes>

legal notes
=================
| SPDX-FileCopyrightText: © 2022 ekvip automation GmbH <info@ekvip.de>
| SPDX-License-Identifier: Apache-2.0
| For details check: Apache-2.0_

.. _Apache-2.0: https://www.apache.org/licenses/LICENSE-2.0

.. </legal notes>

*)
PROPERTY object : CNM_CollectionInterfaces.CNM_AbstractObject.IObject
GET
object := THIS^.dataObject;
END_GET
SET
THIS^.dataObject := object;
END_SET
END_PROPERTY


(*

## Short summary

This property returns the previous element that is linked to this element. Previous element next should be this object.
Previous is not 

.. <legal notes>

legal notes
=================
| SPDX-FileCopyrightText: © 2022 ekvip automation GmbH <info@ekvip.de>
| SPDX-License-Identifier: Apache-2.0
| For details check: Apache-2.0_

.. _Apache-2.0: https://www.apache.org/licenses/LICENSE-2.0

.. </legal notes>

*)
PROPERTY previous : CNM_CollectionInterfaces.IDoublyLinkedElement
GET
previous := THIS^.previousElement;
END_GET
SET
THIS^.previousElement := previous;
END_SET
END_PROPERTY

END_FUNCTION_BLOCK

// ---- Collection/classes/ForEachStrategyExecutor.TcPOU
(*

## Short summary

An class to implement parallel and serial foreach strategies.

**Warning:**
Uses the iterate function of the attached collection and will thus conflict with other 
foreach and iterate statements of the same collection instance.



.. <legal notes>

legal notes
=================
| SPDX-FileCopyrightText: © 2024 ekvip automation GmbH <info@ekvip.de>
| SPDX-License-Identifier: Apache-2.0
| For details check: Apache-2.0_

.. _Apache-2.0: https://www.apache.org/licenses/LICENSE-2.0

.. </legal notes>



*)
FUNCTION_BLOCK INTERNAL FINAL ForEachStrategyExecutor EXTENDS CNM_AbstractObject.Object IMPLEMENTS CNM_CollectionInterfaces.IForEachStrategy
VAR
	usedCollection :CNM_CollectionInterfaces.ICollection;
	{attribute 'no_copy'}
	serialIterator :CNM_CollectionInterfaces.IIterator;
	{attribute 'no_copy'}
	parallelIterator :CNM_CollectionInterfaces.IIterator;
	{attribute 'no_Copy'}
	instantExecutor  :ForEachInstantStrategyExecutor(THIS^.usedCollection);
END_VAR

(*

## Short summary

This abstract property returns the class name of the concrete object, 
which is useful to check the class name for ``__DELETE``.

.. <legal notes>

legal notes
=================
| SPDX-FileCopyrightText: © 2022 ekvip automation GmbH <info@ekvip.de>
| SPDX-License-Identifier: Apache-2.0
| For details check: Apache-2.0_

.. _Apache-2.0: https://www.apache.org/licenses/LICENSE-2.0

.. </legal notes>

*)

PROPERTY className :CNM_AbstractObject.ClassName
GET
className := 'CNM_Collections.ForEachStrategyExecutor';
END_GET
END_PROPERTY

(*

## Short summary

Mark the object as deleted, as it staiys in the memory.

.. <legal notes>

legal notes
=================
| SPDX-FileCopyrightText: © 2022 ekvip automation GmbH <info@ekvip.de>
| SPDX-License-Identifier: Apache-2.0
| For details check: Apache-2.0_

.. _Apache-2.0: https://www.apache.org/licenses/LICENSE-2.0

.. </legal notes>

*)
METHOD FB_Exit : BOOL
VAR_INPUT
	(* TRUE: the exit method is called in order to leave the instance which will be copied afterwards (online change).*)
	bInCopyCode	: BOOL;
END_VAR
IF(THIS^.isObjectValid(THIS^.serialIterator))THEN
	THIS^.serialIterator.destruct();
	THIS^.serialIterator := 0;
END_IF
IF(THIS^.isObjectValid(THIS^.parallelIterator))THEN
	THIS^.parallelIterator.destruct();
	THIS^.parallelIterator := 0;
END_IF
END_METHOD

//FB_Init is always available implicitly and it is used primarily for initialization.
//The return value is not evaluated. For a specific influence, you can also declare the
//methods explicitly and provide additional code there with the standard initialization
//code. You can evaluate the return value.
METHOD FB_Init: BOOL
VAR_INPUT
    bInitRetains: BOOL; // TRUE: the retain variables are initialized (reset warm / reset cold)
    bInCopyCode: BOOL;  // TRUE: the instance will be copied to the copy code afterward (online change)   
	collection : CNM_CollectionInterfaces.ICollection;
END_VAR
usedCollection := collection;
THIS^.instantExecutor.attachCollection(collection);
END_METHOD

(*

## Short summary

This property returns a fluent interface for immediate (wihtin one call) operations of appliers.

.. <legal notes>

legal notes
=================
| SPDX-FileCopyrightText: © 2025 ekvip automation GmbH <info@ekvip.de>
| SPDX-License-Identifier: Apache-2.0
| For details check: Apache-2.0_

.. _Apache-2.0: https://www.apache.org/licenses/LICENSE-2.0

.. </legal notes>



*)

PROPERTY instant : CNM_CollectionInterfaces.IInstantForEachStrategy
GET
instant := THIS^.instantExecutor;
END_GET
END_PROPERTY

(*

## Short summary

Method to perform a given action on all objects inside the collection.
All objects are invoked with the applier each cycle until all are done.
Needs to reset the execution flag between calls.
If at any point the applier returns an error the foreach stops and returns an error.
Action to perform needs to implement `IApplier`.
**Example:**
You have a list of numbers: 1 2 3 and a ConcreteIncrementApplier that can take  a number and increment it. 
Calling ```list.forEach(TRUE, ConcreteIncrementApplier)``` will increment all numbers in the list, becoming: 2 3 4.

**Example 2:**
```
myIntCollectionInstance.foreach.parallel(execute := false);
myIntCollectionInstance.foreach.parallel(execute := true, applier := double);
```

.. <legal notes>

legal notes
=================
| SPDX-FileCopyrightText: © 2025 ekvip automation GmbH <info@ekvip.de>
| SPDX-License-Identifier: Apache-2.0
| For details check: Apache-2.0_

.. _Apache-2.0: https://www.apache.org/licenses/LICENSE-2.0

.. </legal notes>


**Return:** CNM_ReturnTypes.ExecutionState

*)
METHOD parallel : CNM_ReturnTypes.SingleExecutionState
VAR_INPUT
	(*control bit to start or abort the forEach loop*)
	execute	: BOOL;
	(*the applier (action) to be used on all obejcts in the collection*)
	applier	: CNM_CollectionInterfaces.IApplier;
END_VAR
VAR
	continueForeach :BOOL;
	chained			:CNM_CollectionInterfaces.IChainedApplier;
END_VAR
VAR_INST
	object :CNM_AbstractObject.IObject;
	applierIndex 	:UDINT;
	step 			:DINT;
	currentApplier 	:CNM_CollectionInterfaces.IApplier;
	cycleManager	:CNM_CycleManager.SimpleCycleManager;
END_VAR
VAR CONSTANT
	STEP_INIT :DINT := CNM_ReturnTypes.DefaultSteps.STEP.INIT;
	STEP_SELECT_APPLIER :DINT := 2;
	STEP_APPLY :DINT := 3;
	STEP_SUCCESS :DINT := CNM_ReturnTypes.DefaultSteps.STEP.SUCCESS;
	STEP_ERROR :DINT := CNM_ReturnTypes.DefaultSteps.STEP.ERROR;
	NULL : __XWORD := 0;
END_VAR
REPEAT
	continueForeach := FALSE; 
	cycleManager(execute := execute);
	CASE cycleManager.step.current OF
	STEP_INIT:		
		cycleManager.configuration.sequence.requireSuccessStep := FALSE;
		applierIndex := 0;
		currentApplier := 0;
		continueForeach := TRUE;
		cycleManager.proceed();
		cycleManager.step.next := SEL(THIS^.isObjectNull(applier), STEP_SELECT_APPLIER, STEP_ERROR);
		IF ((
			THIS^.isObjectNull(THIS^.parallelIterator)
		) AND_THEN (
			THIS^.usedCollection.createNewIterator(iterator => THIS^.parallelIterator)
			<> CNM_ReturnTypes.SingleExecutionResult.SUCCESS
		)
	) THEN
		cycleManager.step.next := STEP_ERROR;
	END_IF
		
	STEP_SELECT_APPLIER:
		continueForeach := TRUE;
		step :=  THIS^.selectApplier(
			nextStep := STEP_APPLY,
			applier := applier,
			applierIndex := applierIndex,
			nextApplier := currentApplier
		);
		IF step = STEP_SUCCESS THEN
			cycleManager.proceedWith(STEP_SUCCESS);
		ELSE
			THIS^.parallelIterator.iterate(FALSE);
			WHILE( 
				THIS^.parallelIterator.iterate(execute := TRUE, object => object) 
				= CNM_ReturnTypes.SingleExecutionState.BUSY
			)DO
				IF(currentApplier.accept(object) = CNM_ReturnTypes.SingleExecutionResult.SUCCESS)THEN	
					currentApplier.apply(FALSE);
					CONTINUE;
				END_IF
				cycleManager.step.next := STEP_ERROR;
				EXIT;
			END_WHILE
			cycleManager.proceed();
		END_IF
	STEP_APPLY: 
		cycleManager.step.next := STEP_SELECT_APPLIER;
		THIS^.parallelIterator.iterate(FALSE);
		WHILE( 	
			THIS^.parallelIterator.iterate(execute := TRUE, object => object) 
			= CNM_ReturnTypes.SingleExecutionState.BUSY
		)DO
			currentApplier.accept(object);
			CASE (currentApplier.apply(TRUE)) OF
			CNM_ReturnTypes.SingleExecutionState.BUSY: 
				cycleManager.step.next := STEP_APPLY;
			CNM_ReturnTypes.SingleExecutionState.SUCCESS:; 
			ELSE
				continueForeach := TRUE;
				cycleManager.step.next := STEP_ERROR; 
				EXIT;
			END_CASE
		END_WHILE
		cycleManager.proceed();
	END_CASE
UNTIL (NOT continueForeach OR_ELSE NOT execute)
END_REPEAT

parallel := cycleManager.state;
END_METHOD

METHOD PRIVATE selectApplier : DINT
VAR_INPUT
	nextStep : DINT;
	applier : CNM_CollectionInterfaces.IApplier;
END_VAR
VAR_IN_OUT
	applierIndex : UDINT;
	nextApplier :CNM_CollectionInterfaces.IApplier;
END_VAR
VAR
	chained	:CNM_CollectionInterfaces.IChainedApplier;
END_VAR
VAR CONSTANT
	NULL : __XWORD := 0;
END_VAR
selectApplier := CNM_ReturnTypes.DefaultSteps.STEP.SUCCESS;
IF (__QUERYINTERFACE(applier, chained) AND_THEN (chained.actions.count > applierIndex)) THEN
	nextApplier := chained.actions.getApplier(index := applierIndex);
	selectApplier := nextStep;
	applierIndex := (applierIndex + 1);
ELSIF (THIS^.isObjectNull(nextApplier)) THEN
	nextApplier := applier;	
	selectApplier := nextStep;
END_IF
END_METHOD

(*

## Short summary

Method to perform a given action on all objects inside the collection.
Objects are invoked with the applier in order until the applier returns 'SUCCESS', 
only then the next object will be invoked.
When an applier returns BUSY, foreach won't continue on the next object and returns BUSY.
The order in which the appliers are invoked on the objects is defined by the iterator.
If at any point the applier returns an error the serial foreach stops and returns an error.

.. <legal notes>

legal notes
=================
| SPDX-FileCopyrightText: © 2022 ekvip automation GmbH <info@ekvip.de>
| SPDX-License-Identifier: Apache-2.0
| For details check: Apache-2.0_

.. _Apache-2.0: https://www.apache.org/licenses/LICENSE-2.0

.. </legal notes>


**Return:** ``SUCCESS``: if applier returned SUCCESS on every object,
    ``ABORTED``: execute has a falling edge during iterate,
    ``BUSY``: When serial had rising edge on execute and applier returned busy for last evaluated object,
    ``IDLE``: serial wasn't started yet,
	``ERROR``: error occured during execution

*)

METHOD serial : CNM_ReturnTypes.SingleExecutionState
VAR_INPUT
	(*control bit to start or abort the forEach loop*)
	execute	: BOOL;
	(*the applier (action) to be used on all obejcts in the collection*)
	applier	: CNM_CollectionInterfaces.IApplier;
END_VAR
VAR
	continueForeach :BOOL;
END_VAR
VAR_INST
	object :CNM_AbstractObject.IObject;
	applierIndex 	:UDINT;
	returnState 	:CNM_ReturnTypes.SingleExecutionState := CNM_ReturnTypes.SingleExecutionState.IDLE;;
	returnStateObjects 	:CNM_ReturnTypes.SingleExecutionState;
	returnStateApply 	:CNM_ReturnTypes.SingleExecutionState;
	currentApplier 	:CNM_CollectionInterfaces.IApplier;
	cycleManager 	:CNM_CycleManager.SimpleCycleManager;
END_VAR
VAR CONSTANT
	STEP_IDLE :DINT := CNM_ReturnTypes.DefaultSteps.STEP.IDLE;
	STEP_INIT :DINT := CNM_ReturnTypes.DefaultSteps.STEP.INIT;
	STEP_SELECT_APPLIER :DINT := 2;
	STEP_GET_OBJECT :DINT := 3;
	STEP_APPLY :DINT := 4;
	STEP_SUCCESS :DINT := CNM_ReturnTypes.DefaultSteps.STEP.SUCCESS;
	STEP_ERROR :DINT := CNM_ReturnTypes.DefaultSteps.STEP.ERROR;
	STEP_ABORT :DINT := CNM_ReturnTypes.DefaultSteps.STEP.ABORT;
	
	NULL : __XWORD := 0;
END_VAR
REPEAT
	continueForeach := FALSE;
	cycleManager(execute := execute);
	CASE cycleManager.step.current OF
	STEP_INIT:
		cycleManager.configuration.sequence.requireSuccessStep := FALSE;
		applierIndex := 0;
		currentApplier := 0;
		continueForeach := TRUE;
		cycleManager.step.next := SEL(THIS^.isObjectNull(applier), STEP_SELECT_APPLIER, STEP_ERROR);
		IF ((
				THIS^.isObjectNull(THIS^.serialIterator)
			) AND_THEN (
				THIS^.usedCollection.createNewIterator(iterator => THIS^.serialIterator)
				<> CNM_ReturnTypes.SingleExecutionResult.SUCCESS
			)
		) THEN
			cycleManager.step.next := STEP_ERROR;
		END_IF
		cycleManager.proceed();
		
	STEP_SELECT_APPLIER:
		continueForeach := TRUE;
		THIS^.serialIterator.iterate(execute := FALSE);
		cycleManager.proceedWith(
			step := THIS^.selectApplier(
				nextStep := STEP_GET_OBJECT,
				applier := applier,
				applierIndex := applierIndex,
				nextApplier := currentApplier
			)
		);
		
	STEP_GET_OBJECT: 
		returnStateObjects := THIS^.serialIterator.iterate(execute := TRUE, object => object);			
		CASE (returnStateObjects) OF
		CNM_ReturnTypes.SingleExecutionState.BUSY:
			IF(currentApplier.accept(object) = CNM_ReturnTypes.SingleExecutionResult.SUCCESS)THEN	
				currentApplier.apply(FALSE);					
				cycleManager.step.next := STEP_APPLY;
			ELSE
				cycleManager.step.next := STEP_ERROR; 
			END_IF
		CNM_ReturnTypes.SingleExecutionState.SUCCESS:
			cycleManager.step.next := STEP_SELECT_APPLIER; 
		CNM_ReturnTypes.SingleExecutionState.ABORTED:
			cycleManager.step.next := STEP_ABORT; 
		ELSE
			cycleManager.step.next := STEP_ERROR; 
		END_CASE
		continueForeach := TRUE;
		cycleManager.proceed();
		
	STEP_APPLY: 	
		continueForeach := TRUE;
		IF(currentApplier.accept(object) = CNM_ReturnTypes.SingleExecutionResult.SUCCESS)THEN				
			returnStateApply := currentApplier.apply(TRUE);
			CASE (returnStateApply) OF
			CNM_ReturnTypes.SingleExecutionState.BUSY:
				continueForeach := FALSE;
			CNM_ReturnTypes.SingleExecutionState.SUCCESS:
				cycleManager.proceedWith(STEP_GET_OBJECT); 
			CNM_ReturnTypes.SingleExecutionState.ABORTED:
				cycleManager.proceedWith(STEP_ABORT); 
			ELSE
				cycleManager.proceedWith(STEP_ERROR); 
			END_CASE
		ELSE
			cycleManager.proceedWith(STEP_ERROR); 
		END_IF		
	END_CASE
UNTIL (NOT continueForeach)
END_REPEAT
serial := cycleManager.state;
END_METHOD

END_FUNCTION_BLOCK

// ---- Collection/classes/ForEachInstantStrategyExecutor.TcPOU
(*

## Short summary

An class to implement parallel and serial foreach strategies.

**Warning:**
Uses the iterate function of the attached collection and will thus conflict with other 
foreach and iterate statements of the same collection instance.



.. <legal notes>

legal notes
=================
| SPDX-FileCopyrightText: © 2024 ekvip automation GmbH <info@ekvip.de>
| SPDX-License-Identifier: Apache-2.0
| For details check: Apache-2.0_

.. _Apache-2.0: https://www.apache.org/licenses/LICENSE-2.0

.. </legal notes>



*)
FUNCTION_BLOCK INTERNAL FINAL ForEachInstantStrategyExecutor EXTENDS CNM_AbstractObject.Object IMPLEMENTS CNM_CollectionInterfaces.IInstantForEachStrategy
VAR
	usedCollection :CNM_CollectionInterfaces.ICollection;
	{attribute 'no_copy'}
	serialIterator :CNM_CollectionInterfaces.IIterator;
	{attribute 'no_copy'}
	parallelIterator :CNM_CollectionInterfaces.IIterator;
END_VAR

METHOD INTERNAL attachCollection
VAR_INPUT
	collection : CNM_CollectionInterfaces.ICollection;
END_VAR
THIS^.usedCollection := collection;
END_METHOD

(*

## Short summary

This abstract property returns the class name of the concrete object, 
which is useful to check the class name for ``__DELETE``.

.. <legal notes>

legal notes
=================
| SPDX-FileCopyrightText: © 2022 ekvip automation GmbH <info@ekvip.de>
| SPDX-License-Identifier: Apache-2.0
| For details check: Apache-2.0_

.. _Apache-2.0: https://www.apache.org/licenses/LICENSE-2.0

.. </legal notes>

*)

PROPERTY className :CNM_AbstractObject.ClassName
GET
className := 'CNM_Collections.ForEachStrategyExecutor';
END_GET
END_PROPERTY

(*

## Short summary

Mark the object as deleted, as it staiys in the memory.

.. <legal notes>

legal notes
=================
| SPDX-FileCopyrightText: © 2022 ekvip automation GmbH <info@ekvip.de>
| SPDX-License-Identifier: Apache-2.0
| For details check: Apache-2.0_

.. _Apache-2.0: https://www.apache.org/licenses/LICENSE-2.0

.. </legal notes>

*)
METHOD FB_Exit : BOOL
VAR_INPUT
	(* TRUE: the exit method is called in order to leave the instance which will be copied afterwards (online change).*)
	bInCopyCode	: BOOL;
END_VAR
IF(THIS^.isObjectValid(THIS^.serialIterator))THEN
	THIS^.serialIterator.destruct();
	THIS^.serialIterator := 0;
END_IF
IF(THIS^.isObjectValid(THIS^.parallelIterator))THEN
	THIS^.parallelIterator.destruct();
	THIS^.parallelIterator := 0;
END_IF
END_METHOD

//FB_Init is always available implicitly and it is used primarily for initialization.
//The return value is not evaluated. For a specific influence, you can also declare the
//methods explicitly and provide additional code there with the standard initialization
//code. You can evaluate the return value.
METHOD FB_Init: BOOL
VAR_INPUT
    bInitRetains: BOOL; // TRUE: the retain variables are initialized (reset warm / reset cold)
    bInCopyCode: BOOL;  // TRUE: the instance will be copied to the copy code afterward (online change)   
	collection : CNM_CollectionInterfaces.ICollection;
END_VAR
usedCollection := collection;
END_METHOD

(*

## Short summary

Method to perform a given action on all objects inside the collection.
All objects are invoked with the applier until all are done.
If at any point the applier returns an error the foreach stops and returns an error.
Action to perform needs to implement `IApplier`.

**Attention:** This method is single cycle, what means the call waits for all appliers to finish. 
	Therefore none of the appliers should wait for anything (Events/IO/...) 

**Example:**
You have a list of numbers: 1 2 3 and a ConcreteIncrementApplier that can take  a number and increment it. 
Calling ```list.forEach(ConcreteIncrementApplier)``` will increment all numbers in the list, becoming: 2 3 4.

.. <legal notes>

legal notes
=================
| SPDX-FileCopyrightText: © 2022 ekvip automation GmbH <info@ekvip.de>
| SPDX-License-Identifier: Apache-2.0
| For details check: Apache-2.0_

.. _Apache-2.0: https://www.apache.org/licenses/LICENSE-2.0

.. </legal notes>


**Return:** ``SUCCESS``: All appliers returned with ``SUCCESS``
	``ERROR``: The applier returned error for at least one object, or any other error occured

*)

METHOD parallel :CNM_ReturnTypes.SingleExecutionResult
VAR_INPUT
	(*the applier (action) to be used on all obejcts in the collection*)
	applier		:CNM_CollectionInterfaces.IApplier;
END_VAR
VAR
	continueForeach :BOOL;
	chained			:CNM_CollectionInterfaces.IChainedApplier;
	allObjectsAppliedWithSuccess :BOOL;
	firstApllierCall :BOOL;
	objectState		:CNM_ReturnTypes.SingleExecutionState;
	currentApplier 	:CNM_CollectionInterfaces.IApplier;
	object :CNM_AbstractObject.IObject;
	applierIndex 	:UDINT;
END_VAR
VAR CONSTANT
	NULL : __XWORD := 0;
END_VAR
applierIndex := 0;
currentApplier := 0;
continueForeach := TRUE;
IF ((
		THIS^.isObjectNull(THIS^.parallelIterator)
	) AND_THEN (
		THIS^.usedCollection.createNewIterator(iterator => THIS^.parallelIterator)
		<> CNM_ReturnTypes.SingleExecutionResult.SUCCESS
	)
) THEN
	parallel := CNM_ReturnTypes.SingleExecutionResult.ERROR;
	RETURN;
END_IF

WHILE THIS^.selectApplier(applier, applierIndex, currentApplier) DO
	firstApllierCall := TRUE;
	allObjectsAppliedWithSuccess := FALSE;
	THIS^.parallelIterator.iterate(FALSE);	
	WHILE (NOT allObjectsAppliedWithSuccess) DO
		allObjectsAppliedWithSuccess := TRUE;
		THIS^.parallelIterator.iterate(FALSE);
		//	call applier for all objects until all are success  
		WHILE (
			 THIS^.parallelIterator.iterate(execute := TRUE, object => object) 
				= CNM_ReturnTypes.SingleExecutionState.BUSY
		) DO 
			IF(currentApplier.accept(object) = CNM_ReturnTypes.SingleExecutionResult.SUCCESS)THEN
				IF firstApllierCall THEN currentApplier.apply(FALSE); END_IF;
				objectState := 	currentApplier.apply(TRUE);
				CASE objectState OF
				CNM_ReturnTypes.SingleExecutionState.SUCCESS:
					CONTINUE;
				CNM_ReturnTypes.SingleExecutionState.BUSY:
					allObjectsAppliedWithSuccess := FALSE;
					CONTINUE;
				ELSE
					parallel := CNM_ReturnTypes.SingleExecutionResult.ERROR;
					RETURN;	
				END_CASE
			END_IF
			parallel := CNM_ReturnTypes.SingleExecutionResult.ERROR;
			RETURN;
		END_WHILE
		firstApllierCall := FALSE;
	END_WHILE
END_WHILE	
parallel := CNM_ReturnTypes.SingleExecutionResult.SUCCESS;
END_METHOD

METHOD PRIVATE selectApplier :BOOL
VAR_INPUT
	applier : CNM_CollectionInterfaces.IApplier;
END_VAR
VAR_IN_OUT
	applierIndex : UDINT;
	nextApplier :CNM_CollectionInterfaces.IApplier;
END_VAR
VAR
	chained	:CNM_CollectionInterfaces.IChainedApplier;
END_VAR
VAR CONSTANT
	NULL : __XWORD := 0;
END_VAR
selectApplier := FALSE;
IF (__QUERYINTERFACE(applier, chained) AND_THEN (chained.actions.count > applierIndex)) THEN
	nextApplier := chained.actions.getApplier(index := applierIndex);
	selectApplier := TRUE;
	applierIndex := (applierIndex + 1);
ELSIF (THIS^.isObjectNull(nextApplier)) THEN
	nextApplier := applier;	
	selectApplier := TRUE;
END_IF
END_METHOD

(*

## Short summary

Method to perform a given action on all objects inside the collection.
Objects are invoked with the applier in order until done, only then is the next invoked.
Order is defined by the default iterator.
If at any point the applier returns an error the foreach stops and returns an error.
Action to perform needs to implement `IApplier`.

**Attention:** This method is single cycle, what means the call waits for all appliers to finish. 
	Therefore none of the appliers should wait for anything (Events/IO/...) 

**Example:**
You have a list of numbers: 1 2 3 and a ConcreteIncrementApplier that can take  a number and increment it. 
Calling ```list.forEach(ConcreteIncrementApplier)``` will increment all numbers in the list, becoming: 2 3 4.

.. <legal notes>

legal notes
=================
| SPDX-FileCopyrightText: © 2022 ekvip automation GmbH <info@ekvip.de>
| SPDX-License-Identifier: Apache-2.0
| For details check: Apache-2.0_

.. _Apache-2.0: https://www.apache.org/licenses/LICENSE-2.0

.. </legal notes>


**Return:** ``SUCCESS``: Alle appliers returned with ``SUCCESS``
	``ERROR``: The applier returned error for at least one object, or any other error occured

*)

METHOD serial :CNM_ReturnTypes.SingleExecutionResult
VAR_INPUT
	(*the applier to be used on all objects*)
	applier		:CNM_CollectionInterfaces.IApplier;
END_VAR
VAR
	continueForeach :BOOL;
	objectState :CNM_ReturnTypes.SingleExecutionState;
	object		: CNM_AbstractObject.IObject;
	applierIndex 	:UDINT;
	currentApplier 	:CNM_CollectionInterfaces.IApplier;
END_VAR
VAR CONSTANT
	NULL : __XWORD := 0;
END_VAR
applierIndex := 0;
currentApplier := 0;
IF ((
		THIS^.isObjectNull(THIS^.serialIterator)
	) AND_THEN (
		THIS^.usedCollection.createNewIterator(iterator => THIS^.serialIterator)
		<> CNM_ReturnTypes.SingleExecutionResult.SUCCESS
	)
) THEN
	serial := CNM_ReturnTypes.SingleExecutionResult.ERROR;
	RETURN;
END_IF

WHILE THIS^.selectApplier(applier, applierIndex, currentApplier) DO
	THIS^.serialIterator.iterate(execute := FALSE);
	WHILE (THIS^.serialIterator.iterate(execute := TRUE, object => object) = CNM_ReturnTypes.SingleExecutionState.BUSY) DO
		IF currentApplier.accept(object) <> CNM_ReturnTypes.SingleExecutionResult.SUCCESS THEN
			serial := CNM_ReturnTypes.SingleExecutionResult.ERROR;
			RETURN;
		END_IF
		currentApplier.apply(FALSE);
		WHILE TRUE DO
			objectState := currentApplier.apply(TRUE);
			CASE objectState OF
			CNM_ReturnTypes.SingleExecutionState.SUCCESS:
				EXIT;
			CNM_ReturnTypes.SingleExecutionState.BUSY:
				;
			ELSE
				serial := CNM_ReturnTypes.SingleExecutionResult.ERROR;
				RETURN;
			END_CASE
		END_WHILE
	END_WHILE
END_WHILE

serial := CNM_ReturnTypes.SingleExecutionResult.SUCCESS;
END_METHOD

END_FUNCTION_BLOCK

// ---- Lists/classes/SortingStrategyExecutor.TcPOU
FUNCTION_BLOCK SortingStrategyExecutor EXTENDS CNM_AbstractObject.Object IMPLEMENTS CNM_CollectionInterfaces.ISortable
VAR
	usedList :IListHelpers;
	instantStrategy :InstantSortingStrategyExecutor(THIS^.usedList);
END_VAR

(*

## Short summary

This method sorts the data structure. 
This can take many cycles and should be called until the CNM_ReturnTypes.ExecutionState is no longer ``BUSY``.
Uses the passed comparator or compareTo of the contained objects if no comparator is passed.

.. <legal notes>

legal notes
=================
| SPDX-FileCopyrightText: © 2022 ekvip automation GmbH <info@ekvip.de>
| SPDX-License-Identifier: Apache-2.0
| For details check: Apache-2.0_

.. _Apache-2.0: https://www.apache.org/licenses/LICENSE-2.0

.. </legal notes>


**Return:** ``ABORTED``: While sort was pending,execute had a falling edge,
	``BUSY``: Sort is in progress
	``ERROR``: Sort was not able to finish (p.e. List changed) call sort(false) to reset
	``IDLE``: Currently no sort in progress
	``SUCCESS``: Sorting was finished 

*)
METHOD ascending : CNM_CollectionInterfaces.CNM_ReturnTypes.SingleExecutionState
VAR_INPUT
	(*control bit to start or abort the sorting, needs to be active until the ExecutionState is SUCCESS*)
	execute	: BOOL;
	(*Optional: the comparator that should be used for the sort. Must not be changed while sort is in process*)
	comparator	: CNM_CollectionInterfaces.CNM_AbstractObject.IComparator := 0;
END_VAR
ascending := THIS^.usedList.sorting(
	execute := execute,
	order := SortingOrder.ASCENDING,
	comparator := comparator
);
END_METHOD

PROPERTY className : CNM_AbstractObject.ClassName
GET
className := 'CNM_Collections.SortingStrategyExecutor';
END_GET
END_PROPERTY

(*

## Short summary

This method sorts the Sortable in the inverted order, so from great to low
Result of the passed comparator is inverted. If no comparator is passed, compareTo of the Objects is used (inverted)


.. <legal notes>

legal notes
=================
| SPDX-FileCopyrightText: © 2022 ekvip automation GmbH <info@ekvip.de>
| SPDX-License-Identifier: Apache-2.0
| For details check: Apache-2.0_

.. _Apache-2.0: https://www.apache.org/licenses/LICENSE-2.0

.. </legal notes>


**Return:** ``ABORTED``: While inverseSort was pending,execute had a falling edge,
	``BUSY``: inverseSort is in progress
	``ERROR``: inverseSort was not able to finish (p.e. List changed) call inverseSort(false) to reset
	``SUCCESS``: Inversing was finished 
*)
METHOD descending : CNM_CollectionInterfaces.CNM_ReturnTypes.SingleExecutionState
VAR_INPUT
	(*control bit to start or abort the inverting, needs to be active until the ExecutionState is noz longer busy*)
	execute	: BOOL;
	(*the comparator that should be used for the sort. Must not be changed while sort is in process*)
	comparator	: CNM_CollectionInterfaces.CNM_AbstractObject.IComparator := 0;
END_VAR
descending := THIS^.usedList.sorting(
	execute := execute,
	order := SortingOrder.DESCENDING,
	comparator := comparator
);
END_METHOD

(*

## Short summary

The constructor ``FB_init`` is needed to create an unique hash code.
The hash code is a pseudo random number create with a [xorshift](https://en.wikipedia.org/wiki/Xorshift) algorithm.
It can be overwritten on derivations, because it will be called implicit, ``SUPER^.FB_init()`` is not required.
For more information check: [Behavoir with derived function blocks](https://infosys.beckhoff.com/content/1033/tc3_plc_intro/5482088715.html?id=6983869892358031022).

.. <legal notes>

legal notes
=================
| SPDX-FileCopyrightText: © 2022 ekvip automation GmbH <info@ekvip.de>
| SPDX-License-Identifier: Apache-2.0
| For details check: Apache-2.0_

.. _Apache-2.0: https://www.apache.org/licenses/LICENSE-2.0

.. </legal notes>



*)
METHOD FB_init : BOOL
VAR_INPUT
	(* if TRUE, the retain variables are initialized (warm start / cold start)*)
	bInitRetains	: BOOL;
	(* if TRUE, the instance afterwards gets moved into the copy code (online change) *)
	bInCopyCode	: BOOL;
	(* the list it should be attached to *)
	list :IListHelpers;
END_VAR
THIS^.usedList := list;
THIS^.instantStrategy.attachList(list);
END_METHOD

(*

## Short summary

This property returns a fluent interface for immediate sorting operations that will finish wihtin one call.

.. <legal notes>

legal notes
=================
| SPDX-FileCopyrightText: © 2025 ekvip automation GmbH <info@ekvip.de>
| SPDX-License-Identifier: Apache-2.0
| For details check: Apache-2.0_

.. _Apache-2.0: https://www.apache.org/licenses/LICENSE-2.0

.. </legal notes>



*)
PROPERTY instant : CNM_CollectionInterfaces.IInstantSortable
GET
instant := THIS^.instantStrategy;
END_GET
END_PROPERTY

END_FUNCTION_BLOCK

// ---- Lists/classes/InstantSortingStrategyExecutor.TcPOU
FUNCTION_BLOCK InstantSortingStrategyExecutor EXTENDS CNM_AbstractObject.Object IMPLEMENTS CNM_CollectionInterfaces.IInstantSortable
VAR
	usedList :IListHelpers;
END_VAR

(*
## Short summary

This method sorts the data structure immediately in an ascending order. 
The sorting will be finished within method call.
Uses the passed comparator or compareTo of the contained objects if no comparator is passed.

.. <legal notes>

legal notes
=================
| SPDX-FileCopyrightText: © 2025 ekvip automation GmbH <info@ekvip.de>
| SPDX-License-Identifier: Apache-2.0
| For details check: Apache-2.0_

.. _Apache-2.0: https://www.apache.org/licenses/LICENSE-2.0

.. </legal notes>


**Return:** ``ABORTED``: While sort was pending,execute had a falling edge,
	``ERROR``: Sort was not able to finish (p.e. List changed) call sort(false) to reset
	``SUCCESS``: Sorting was finished 

*)

METHOD ascending : CNM_CollectionInterfaces.CNM_ReturnTypes.SingleExecutionResult
VAR_INPUT
	(*Optional: the comparator that should be used for the sort. Must not be changed while sort is in process*)
	comparator	: CNM_CollectionInterfaces.CNM_AbstractObject.IComparator := 0;
END_VAR
ascending := THIS^.usedList.instantSorting(
	order := SortingOrder.ASCENDING,
	comparator := comparator
);
END_METHOD

METHOD INTERNAL attachList
VAR_INPUT
	list :IListHelpers;
END_VAR
THIS^.usedList := list;
END_METHOD

PROPERTY className : CNM_AbstractObject.ClassName
GET
className := 'CNM_Collections.InstantSortingStrategyExecutor';
END_GET
END_PROPERTY

(*

## Short summary

This method sorts the data structure in a descending order, so from great to low.
The sorting will be finished within method call.
Uses the passed comparator or compareTo of the contained objects if no comparator is passed.

.. <legal notes>

legal notes
=================
| SPDX-FileCopyrightText: © 2022 ekvip automation GmbH <info@ekvip.de>
| SPDX-License-Identifier: Apache-2.0
| For details check: Apache-2.0_

.. _Apache-2.0: https://www.apache.org/licenses/LICENSE-2.0

.. </legal notes>


**Return:** ``ABORTED``: While inverseSort was pending,execute had a falling edge,
	``ERROR``: inverseSort was not able to finish (p.e. List changed) call inverseSort(false) to reset
	``SUCCESS``: Inversing was finished 
*)

METHOD descending :CNM_ReturnTypes.SingleExecutionResult
VAR_INPUT
	(*the comparator that should be used for the sort. Must not be changed while sort is in process*)
	comparator :CNM_AbstractObject.IComparator := 0;
END_VAR
descending := THIS^.usedList.instantSorting(
	order := SortingOrder.DESCENDING,
	comparator := comparator
);
END_METHOD

(*

## Short summary

The constructor ``FB_init`` is needed to create an unique hash code.
The hash code is a pseudo random number create with a [xorshift](https://en.wikipedia.org/wiki/Xorshift) algorithm.
It can be overwritten on derivations, because it will be called implicit, ``SUPER^.FB_init()`` is not required.
For more information check: [Behavoir with derived function blocks](https://infosys.beckhoff.com/content/1033/tc3_plc_intro/5482088715.html?id=6983869892358031022).

.. <legal notes>

legal notes
=================
| SPDX-FileCopyrightText: © 2022 ekvip automation GmbH <info@ekvip.de>
| SPDX-License-Identifier: Apache-2.0
| For details check: Apache-2.0_

.. _Apache-2.0: https://www.apache.org/licenses/LICENSE-2.0

.. </legal notes>



*)
METHOD FB_init : BOOL
VAR_INPUT
	(* if TRUE, the retain variables are initialized (warm start / cold start)*)
	bInitRetains	: BOOL;
	(* if TRUE, the instance afterwards gets moved into the copy code (online change) *)
	bInCopyCode	: BOOL;
	(* the list it should be attached to *)
	list :IListHelpers;
END_VAR
THIS^.usedList := list;
END_METHOD

END_FUNCTION_BLOCK

// ---- Lists/ArrayList/ArrayListIterator/classes/ForwardArrayListIterator.TcPOU
(*

## Short summary

This class can be used as a simple iterator for array lists. It iterates from first element to last element.

.. <legal notes>

legal notes
=================
| SPDX-FileCopyrightText: © 2024 ekvip automation GmbH <info@ekvip.de>
| SPDX-License-Identifier: Apache-2.0
| For details check: Apache-2.0_

.. _Apache-2.0: https://www.apache.org/licenses/LICENSE-2.0

.. </legal notes>



*)

{attribute 'enable_dynamic_creation'}
FUNCTION_BLOCK ForwardArrayListIterator EXTENDS AbstractArrayListIterator

PROPERTY className :CNM_AbstractObject.ClassName
GET
className := 'ForwardArrayListIterator';
END_GET
END_PROPERTY

(*

## Short summary

The constructor ``FB_init`` is needed to create an unique hash code.
The hash code is a pseudo random number create with a [xorshift](https://en.wikipedia.org/wiki/Xorshift) algorithm.
It can be overwritten on derivations, because it will be called implicit, ``SUPER^.FB_init()`` is not required.
For more information check: [Behavoir with derived function blocks](https://infosys.beckhoff.com/content/1033/tc3_plc_intro/5482088715.html?id=6983869892358031022).

.. <legal notes>

legal notes
=================
| SPDX-FileCopyrightText: © 2022 ekvip automation GmbH <info@ekvip.de>
| SPDX-License-Identifier: Apache-2.0
| For details check: Apache-2.0_

.. _Apache-2.0: https://www.apache.org/licenses/LICENSE-2.0

.. </legal notes>



*)
METHOD FB_init : BOOL
VAR_INPUT
	(* if TRUE, the retain variables are initialized (warm start / cold start)*)
	bInitRetains	: BOOL;
	(* if TRUE, the instance afterwards gets moved into the copy code (online change) *)
	bInCopyCode	: BOOL;
	(* the array list which should be iterated, can be 0 *)
	arrayList :REFERENCE TO ArrayList;
END_VAR
THIS^.direction := IterationDirection.FORWARD;
END_METHOD

END_FUNCTION_BLOCK

// ---- Lists/ArrayList/ArrayListIterator/classes/AbstractArrayListIterator.TcPOU
(*

## Short summary

An abstract class to implement the basic datastructure dependency to array lists.

.. <legal notes>

legal notes
=================
| SPDX-FileCopyrightText: © 2024 ekvip automation GmbH <info@ekvip.de>
| SPDX-License-Identifier: Apache-2.0
| For details check: Apache-2.0_

.. _Apache-2.0: https://www.apache.org/licenses/LICENSE-2.0

.. </legal notes>



*)

FUNCTION_BLOCK ABSTRACT AbstractArrayListIterator EXTENDS AbstractIterator IMPLEMENTS IArrayListIterator
VAR	
	{attribute 'hide'}
	list 			:REFERENCE TO ArrayList;
	nextIndex 		:__XWORD;
	direction 		:IterationDirection;
END_VAR

(*

## Short summary

This method attaches an array list to the iterator.

.. <legal notes>

legal notes
=================
| SPDX-FileCopyrightText: © 2024 ekvip automation GmbH <info@ekvip.de>
| SPDX-License-Identifier: Apache-2.0
| For details check: Apache-2.0_

.. _Apache-2.0: https://www.apache.org/licenses/LICENSE-2.0

.. </legal notes>

*)

METHOD attachArrayList
VAR_INPUT
	(* The list to be attached. Should be a reference of type ``ArrayList`` *)
	list :REFERENCE TO ArrayList;
END_VAR
THIS^.list REF= list;
THIS^.reset();
END_METHOD

(*

## Short summary

The constructor ``FB_init`` is needed to create an unique hash code.
The hash code is a pseudo random number create with a [xorshift](https://en.wikipedia.org/wiki/Xorshift) algorithm.
It can be overwritten on derivations, because it will be called implicit, ``SUPER^.FB_init()`` is not required.
For more information check: [Behavoir with derived function blocks](https://infosys.beckhoff.com/content/1033/tc3_plc_intro/5482088715.html?id=6983869892358031022).

.. <legal notes>

legal notes
=================
| SPDX-FileCopyrightText: © 2022 ekvip automation GmbH <info@ekvip.de>
| SPDX-License-Identifier: Apache-2.0
| For details check: Apache-2.0_

.. _Apache-2.0: https://www.apache.org/licenses/LICENSE-2.0

.. </legal notes>



*)
METHOD FB_init : BOOL
VAR_INPUT
	(* if TRUE, the retain variables are initialized (warm start / cold start)*)
	bInitRetains	:BOOL;
	(* if TRUE, the instance afterwards gets moved into the copy code (online change) *)
	bInCopyCode	:BOOL;
	(* the array list which should be iterated, can be 0 *)
	arrayList :REFERENCE TO ArrayList;
END_VAR
THIS^.list REF= arrayList;
END_METHOD

(*

## Short summary

This method returns if there exists another element to iterate to.

**Example:**
```
WHILE(iterator.hasNext())DO
	iterator.getNext().name;
END_WHILE
```

.. <legal notes>

legal notes
=================
| SPDX-FileCopyrightText: © 2022 ekvip automation GmbH <info@ekvip.de>
| SPDX-License-Identifier: Apache-2.0
| For details check: Apache-2.0_

.. _Apache-2.0: https://www.apache.org/licenses/LICENSE-2.0

.. </legal notes>


**Return:** ``TRUE``: Iterator has a next object that can be fetched with getNext()
	``FALSE``: Iterator finished

*)

METHOD hasNext :BOOL
hasNext := THIS^.isObjectValid(THIS^.list) AND_THEN (THIS^.nextIndex < THIS^.list.size);
END_METHOD

(*

## Short summary

This method returns the next object in the iteration and returns an execution state.
**Example:**
You have a list: 1 2 3
the first iterate call will return CNM_ReturnTypes.BUSY and object = 1
the second iterate call will return CNM_ReturnTypes.BUSY and object = 2
the third iterate call will return CNM_ReturnTypes.BUSY and object = 3
the forth iterate call will return CNM_ReturnTypes.SUCCESS and object = NULL

.. <legal notes>

legal notes
=================
| SPDX-FileCopyrightText: © 2022 ekvip automation GmbH <info@ekvip.de>
| SPDX-License-Identifier: Apache-2.0
| For details check: Apache-2.0_

.. _Apache-2.0: https://www.apache.org/licenses/LICENSE-2.0

.. </legal notes>


**Return:** ``SingleExecutionState.SUCCESS``: Iteration finished, no new elements, returned NULL object
    ``SingleExecutionState.ERROR``: error during iteration
    ``SingleExecutionState.ABORT``: iteration aborted
    ``SingleExecutionState.BUSY``: returned an element and iteration in progress	
    ``SingleExecutionState.IDLE``: ready for iteration

*)
METHOD FINAL iterate : CNM_ReturnTypes.SingleExecutionState
VAR_INPUT
	(*control bit to start or abort the iterate (see SingleExecutionState)*)
	execute	: BOOL;
END_VAR
VAR_OUTPUT
	(*the returned object of the iteration*)
	object :CNM_AbstractObject.IObject;
END_VAR
VAR_INST	
	lastChangeVersion :__XWORD;
	cycleManager :CNM_CycleManager.SimpleCycleManager;
END_VAR
VAR CONSTANT
	NULL :__XWORD := 0;
	INIT :DINT := CNM_ReturnTypes.DefaultSteps.STEP.INIT;
	ITERATING :DINT := INIT + 1;
	ERROR :DINT := CNM_ReturnTypes.DefaultSteps.STEP.ERROR;
	SUCCESS :DINT := CNM_ReturnTypes.DefaultSteps.STEP.SUCCESS;
END_VAR
cycleManager(execute := execute);

CASE cycleManager.step.current OF
INIT:
	cycleManager.configuration.sequence.requireSuccessStep := FALSE;
	THIS^.nextIndex := 0;
	lastChangeVersion := THIS^.list.changesToCollection;
	THIS^.currentObject := 0;
	IF(THIS^.hasNext())THEN
		THIS^.currentObject := THIS^.list.container[SEL((THIS^.direction = IterationDirection.BACKWARD), THIS^.nextIndex, THIS^.list.size-1-THIS^.nextIndex)];
		THIS^.nextIndex := THIS^.nextIndex+1;
		IF(THIS^.isObjectValid(THIS^.currentObject))THEN
			cycleManager.proceed();
		ELSE
			cycleManager.proceedWith(ERROR);				
		END_IF
	ELSE
		THIS^.currentObject := NULL;
		cycleManager.proceedWith(SUCCESS);
	END_IF
ITERATING:
	IF (lastChangeVersion <>  THIS^.list.changesToCollection) THEN
		cycleManager.proceedWith(ERROR);
	ELSIF (THIS^.hasNext())THEN
		THIS^.currentObject := THIS^.list.container[SEL((THIS^.direction = IterationDirection.BACKWARD), THIS^.nextIndex, THIS^.list.size-1-THIS^.nextIndex)];
		THIS^.nextIndex := THIS^.nextIndex+1;
		IF(NOT THIS^.isObjectValid(THIS^.currentObject))THEN
			cycleManager.proceedWith(ERROR);				
		END_IF
	ELSE
		THIS^.currentObject := NULL;
		cycleManager.proceedWith(SUCCESS);
	END_IF
END_CASE

object  := THIS^.currentObject;
iterate := cycleManager.state;
END_METHOD

(*

## Short summary

This method resets the iterator.

